LIN {X 0,Y 395.262,Z 435.098,A -85,B 0,C 180,E1 17057.331,E2 17057.331} C_VEL
LIN {X 0,Y 390.739,Z 495.427,A -85,B 0,C 180,E1 17055.904,E2 17055.904} C_VEL
LIN {X 0,Y 384.657,Z 560.923,A -85,B 0,C 180,E1 17054.093,E2 17054.093} C_VEL
LIN {X 0,Y 381.336,Z 596.706,A -85,B 0,C 180,E1 17052.908,E2 17052.908} C_VEL
LIN {X 0,Y 379.095,Z 616.56,A -85,B 0,C 180,E1 17051.979,E2 17051.979} C_VEL
LIN {X 0,Y 376.209,Z 636.469,A -85,B 0,C 180,E1 17050.759,E2 17050.759} C_VEL
LIN {X 0,Y 372.83,Z 655.705,A -85,B 0,C 180,E1 17049.265,E2 17049.265} C_VEL
LIN {X 0,Y 369.199,Z 673.643,A -85,B 0,C 180,E1 17047.542,E2 17047.542} C_VEL
LIN {X 0,Y 365.244,Z 691.251,A -85,B 0,C 180,E1 17045.476,E2 17045.476} C_VEL
LIN {X 0,Y 361.397,Z 707.145,A -85,B 0,C 180,E1 17043.216,E2 17043.216} C_VEL
LIN {X 0,Y 357.759,Z 721.542,A -85,B 0,C 180,E1 17040.76,E2 17040.76} C_VEL
LIN {X 0,Y 354.442,Z 734.528,A -85,B 0,C 180,E1 17038.106,E2 17038.106} C_VEL
LIN {X 0,Y 353.671,Z 737.462,A -85,B 0,C 180,E1 17037.421,E2 17037.421} C_VEL
LIN {X 0,Y 351.666,Z 741.92,A -85,B 0,C 180,E1 17036.434,E2 17036.434} C_VEL
LIN {X 0,Y 343.491,Z 752.769,A -85,B 0,C 180,E1 17033.979,E2 17033.979} C_VEL
LIN {X 0,Y 341.66,Z 756.437,A -85,B 0,C 180,E1 17032.885,E2 17032.885} C_VEL
LIN {X 0,Y 339.571,Z 765.333,A -85,B 0,C 180,E1 17029.568,E2 17029.568} C_VEL
LIN {X 0,Y 338.136,Z 772.212,A -85,B 0,C 180,E1 17026.315,E2 17026.315} C_VEL
LIN {X 0,Y 337.239,Z 777.506,A -85,B 0,C 180,E1 17023.022,E2 17023.022} C_VEL
LIN {X 0,Y 336.721,Z 781.379,A -85,B 0,C 180,E1 17019.572,E2 17019.572} C_VEL
LIN {X 0,Y 336.488,Z 783.588,A -85,B 0,C 180,E1 17016.141,E2 17016.141} C_VEL
LIN {X 0,Y 336.423,Z 784.209,A -85,B 0,C 180,E1 17012.896,E2 17012.896} C_VEL
LIN {X 0,Y 336.482,Z 783.288,A -85,B 0,C 180,E1 17009.489,E2 17009.489} C_VEL
LIN {X 0,Y 336.698,Z 780.724,A -85,B 0,C 180,E1 17006.084,E2 17006.084} C_VEL
LIN {X 0,Y 337.201,Z 776.517,A -85,B 0,C 180,E1 17002.675,E2 17002.675} C_VEL
LIN {X 0,Y 338.065,Z 770.919,A -85,B 0,C 180,E1 16999.434,E2 16999.434} C_VEL
LIN {X 0,Y 339.443,Z 763.662,A -85,B 0,C 180,E1 16996.196,E2 16996.196} C_VEL
LIN {X 0,Y 341.411,Z 754.589,A -85,B 0,C 180,E1 16992.971,E2 16992.971} C_VEL
LIN {X 0,Y 343.953,Z 743.864,A -85,B 0,C 180,E1 16989.878,E2 16989.878} C_VEL
LIN {X 0,Y 347.043,Z 731.447,A -85,B 0,C 180,E1 16986.932,E2 16986.932} C_VEL
LIN {X 0,Y 350.403,Z 718.053,A -85,B 0,C 180,E1 16984.296,E2 16984.296} C_VEL
LIN {X 0,Y 354.037,Z 703.239,A -85,B 0,C 180,E1 16981.859,E2 16981.859} C_VEL
LIN {X 0,Y 357.872,Z 686.847,A -85,B 0,C 180,E1 16979.622,E2 16979.622} C_VEL
LIN {X 0,Y 361.536,Z 669.791,A -85,B 0,C 180,E1 16977.693,E2 16977.693} C_VEL
LIN {X 0,Y 365.122,Z 651.237,A -85,B 0,C 180,E1 16975.977,E2 16975.977} C_VEL
LIN {X 0,Y 368.27,Z 632.306,A -85,B 0,C 180,E1 16974.564,E2 16974.564} C_VEL
LIN {X 0,Y 370.972,Z 612.338,A -85,B 0,C 180,E1 16973.39,E2 16973.39} C_VEL
LIN {X 0,Y 373.069,Z 592.248,A -85,B 0,C 180,E1 16972.505,E2 16972.505} C_VEL
LIN {X 0,Y 377.322,Z 546.729,A -85,B 0,C 180,E1 16971.047,E2 16971.047} C_VEL
LIN {X 0,Y 382.861,Z 484.443,A -85,B 0,C 180,E1 16969.345,E2 16969.345} C_VEL
LIN {X 0,Y 387.038,Z 425.627,A -85,B 0,C 180,E1 16967.978,E2 16967.978} C_VEL
LIN {X 0,Y 389.904,Z 364.859,A -85,B 0,C 180,E1 16966.743,E2 16966.743} C_VEL
LIN {X 0,Y 386.088,Z 359.453,A -85,B 0,C 180,E1 16965.944,E2 16965.944} C_VEL
LIN {X 0,Y 380.964,Z 347.137,A -85,B 0,C 180,E1 16962.826,E2 16962.826} C_VEL
LIN {X 0,Y 376.081,Z 336.257,A -85,B 0,C 180,E1 16959.649,E2 16959.649} C_VEL
LIN {X 0,Y 371.792,Z 327.479,A -85,B 0,C 180,E1 16956.658,E2 16956.658} C_VEL
LIN {X 0,Y 370.912,Z 327.517,A -85,B 0,C 180,E1 16956.374,E2 16956.374} C_VEL
LIN {X 0,Y 365.817,Z 329.462,A -85,B 0,C 180,E1 16955.029,E2 16955.029} C_VEL
LIN {X 0,Y 361.614,Z 332.459,A -85,B 0,C 180,E1 16954.146,E2 16954.146} C_VEL
LIN {X 0,Y 358.196,Z 335.591,A -85,B 0,C 180,E1 16953.553,E2 16953.553} C_VEL
LIN {X 0,Y 355.928,Z 336.945,A -85,B 0,C 180,E1 16952.918,E2 16952.918} C_VEL
LIN {X 0,Y 353.668,Z 378.738,A -85,B 0,C 180,E1 16948.911,E2 16948.911} C_VEL
LIN {X 0,Y 351.265,Z 423.605,A -85,B 0,C 180,E1 16944.646,E2 16944.646} C_VEL
LIN {X 0,Y 349.262,Z 462.521,A -85,B 0,C 180,E1 16940.969,E2 16940.969} C_VEL
LIN {X 0,Y 348.83,Z 465.633,A -85,B 0,C 180,E1 16940.754,E2 16940.754} C_VEL
LIN {X 0,Y 344.684,Z 603.323,A -85,B 0,C 180,E1 16937.135,E2 16937.135} C_VEL
LIN {X 0,Y 344.407,Z 621.566,A -85,B 0,C 180,E1 16936.464,E2 16936.464} C_VEL
LIN {X 0,Y 343.813,Z 639.774,A -85,B 0,C 180,E1 16935.433,E2 16935.433} C_VEL
LIN {X 0,Y 343.002,Z 656.912,A -85,B 0,C 180,E1 16934.088,E2 16934.088} C_VEL
LIN {X 0,Y 342.154,Z 671.753,A -85,B 0,C 180,E1 16932.568,E2 16932.568} C_VEL
LIN {X 0,Y 341.302,Z 684.893,A -85,B 0,C 180,E1 16930.892,E2 16930.892} C_VEL
LIN {X 0,Y 340.457,Z 697.128,A -85,B 0,C 180,E1 16928.955,E2 16928.955} C_VEL
LIN {X 0,Y 339.765,Z 707.457,A -85,B 0,C 180,E1 16926.931,E2 16926.931} C_VEL
LIN {X 0,Y 339.191,Z 717.119,A -85,B 0,C 180,E1 16924.566,E2 16924.566} C_VEL
LIN {X 0,Y 338.818,Z 725.023,A -85,B 0,C 180,E1 16922.03,E2 16922.03} C_VEL
LIN {X 0,Y 338.66,Z 730.537,A -85,B 0,C 180,E1 16919.662,E2 16919.662} C_VEL
LIN {X 0,Y 338.71,Z 734.833,A -85,B 0,C 180,E1 16916.955,E2 16916.955} C_VEL
LIN {X 0,Y 338.938,Z 736.969,A -85,B 0,C 180,E1 16914.414,E2 16914.414} C_VEL
LIN {X 0,Y 339.382,Z 737.372,A -85,B 0,C 180,E1 16911.85,E2 16911.85} C_VEL
LIN {X 0,Y 340.004,Z 735.908,A -85,B 0,C 180,E1 16909.324,E2 16909.324} C_VEL
LIN {X 0,Y 340.843,Z 732.779,A -85,B 0,C 180,E1 16906.887,E2 16906.887} C_VEL
LIN {X 0,Y 341.921,Z 727.575,A -85,B 0,C 180,E1 16904.394,E2 16904.394} C_VEL
LIN {X 0,Y 343.104,Z 721.104,A -85,B 0,C 180,E1 16902.183,E2 16902.183} C_VEL
LIN {X 0,Y 344.485,Z 712.486,A -85,B 0,C 180,E1 16899.972,E2 16899.972} C_VEL
LIN {X 0,Y 345.876,Z 702.622,A -85,B 0,C 180,E1 16898.007,E2 16898.007} C_VEL
LIN {X 0,Y 347.304,Z 690.717,A -85,B 0,C 180,E1 16896.142,E2 16896.142} C_VEL
LIN {X 0,Y 348.601,Z 677.563,A -85,B 0,C 180,E1 16894.518,E2 16894.518} C_VEL
LIN {X 0,Y 349.742,Z 662.299,A -85,B 0,C 180,E1 16893.056,E2 16893.056} C_VEL
LIN {X 0,Y 350.573,Z 646.797,A -85,B 0,C 180,E1 16891.928,E2 16891.928} C_VEL
LIN {X 0,Y 351.092,Z 630.054,A -85,B 0,C 180,E1 16891.038,E2 16891.038} C_VEL
LIN {X 0,Y 352.008,Z 597.232,A -85,B 0,C 180,E1 16889.859,E2 16889.859} C_VEL
LIN {X 0,Y 358.318,Z 513.728,A -85,B 0,C 180,E1 16887.077,E2 16887.077} C_VEL
LIN {X 0,Y 360.474,Z 491.875,A -85,B 0,C 180,E1 16886.307,E2 16886.307} C_VEL
LIN {X 0,Y 363.78,Z 479.698,A -85,B 0,C 180,E1 16885.515,E2 16885.515} C_VEL
LIN {X 0,Y 366.437,Z 478.721,A -85,B 0,C 180,E1 16885.216,E2 16885.216} C_VEL
LIN {X 0,Y 370.915,Z 475.814,A -85,B 0,C 180,E1 16884.864,E2 16884.864} C_VEL
LIN {X 0,Y 374.886,Z 474.256,A -85,B 0,C 180,E1 16884.45,E2 16884.45} C_VEL
LIN {X 0,Y 377.753,Z 472.722,A -85,B 0,C 180,E1 16884.201,E2 16884.201} C_VEL
LIN {X 0,Y 396.698,Z 464.403,A -85,B 0,C 180,E1 16882.483,E2 16882.483} C_VEL
LIN {X 0,Y 402.924,Z 480.075,A -85,B 0,C 180,E1 16880.192,E2 16880.192} C_VEL
LIN {X 0,Y 407.395,Z 488.925,A -85,B 0,C 180,E1 16878.854,E2 16878.854} C_VEL
LIN {X 0,Y 395.273,Z 512.025,A -85,B 0,C 180,E1 16878.047,E2 16878.047} C_VEL
LIN {X 0,Y 390.931,Z 521.783,A -85,B 0,C 180,E1 16877.657,E2 16877.657} C_VEL
LIN {X 0,Y 386.492,Z 551.571,A -85,B 0,C 180,E1 16877.527,E2 16877.527} C_VEL
LIN {X 0,Y 384.035,Z 573.78,A -85,B 0,C 180,E1 16877.191,E2 16877.191} C_VEL
LIN {X 0,Y 381.047,Z 603.773,A -85,B 0,C 180,E1 16876.316,E2 16876.316} C_VEL
LIN {X 0,Y 377.367,Z 630.176,A -85,B 0,C 180,E1 16875.298,E2 16875.298} C_VEL
LIN {X 0,Y 373.423,Z 655.596,A -85,B 0,C 180,E1 16874.014,E2 16874.014} C_VEL
LIN {X 0,Y 369.301,Z 679.477,A -85,B 0,C 180,E1 16872.494,E2 16872.494} C_VEL
LIN {X 0,Y 364.889,Z 703.359,A -85,B 0,C 180,E1 16870.622,E2 16870.622} C_VEL
LIN {X 0,Y 360.964,Z 723.184,A -85,B 0,C 180,E1 16868.757,E2 16868.757} C_VEL
LIN {X 0,Y 356.93,Z 741.602,A -85,B 0,C 180,E1 16866.632,E2 16866.632} C_VEL
LIN {X 0,Y 353.156,Z 757.77,A -85,B 0,C 180,E1 16864.391,E2 16864.391} C_VEL
LIN {X 0,Y 349.271,Z 773.512,A -85,B 0,C 180,E1 16861.765,E2 16861.765} C_VEL
LIN {X 0,Y 345.911,Z 787.154,A -85,B 0,C 180,E1 16859.052,E2 16859.052} C_VEL
LIN {X 0,Y 342.775,Z 800.117,A -85,B 0,C 180,E1 16855.947,E2 16855.947} C_VEL
LIN {X 0,Y 340.23,Z 811.492,A -85,B 0,C 180,E1 16852.666,E2 16852.666} C_VEL
LIN {X 0,Y 338.223,Z 821.847,A -85,B 0,C 180,E1 16848.977,E2 16848.977} C_VEL
LIN {X 0,Y 337.03,Z 829.629,A -85,B 0,C 180,E1 16845.486,E2 16845.486} C_VEL
LIN {X 0,Y 336.389,Z 835.947,A -85,B 0,C 180,E1 16841.835,E2 16841.835} C_VEL
LIN {X 0,Y 336.186,Z 840.283,A -85,B 0,C 180,E1 16838.38,E2 16838.38} C_VEL
LIN {X 0,Y 336.2,Z 843.205,A -85,B 0,C 180,E1 16834.777,E2 16834.777} C_VEL
LIN {X 0,Y 336.246,Z 844.515,A -85,B 0,C 180,E1 16831.363,E2 16831.363} C_VEL
LIN {X 0,Y 336.242,Z 844.359,A -85,B 0,C 180,E1 16827.955,E2 16827.955} C_VEL
LIN {X 0,Y 336.186,Z 842.807,A -85,B 0,C 180,E1 16824.539,E2 16824.539} C_VEL
LIN {X 0,Y 336.185,Z 839.823,A -85,B 0,C 180,E1 16821.103,E2 16821.103} C_VEL
LIN {X 0,Y 336.464,Z 835.014,A -85,B 0,C 180,E1 16817.471,E2 16817.471} C_VEL
LIN {X 0,Y 337.218,Z 828.492,A -85,B 0,C 180,E1 16813.816,E2 16813.816} C_VEL
LIN {X 0,Y 338.62,Z 819.993,A -85,B 0,C 180,E1 16810.149,E2 16810.149} C_VEL
LIN {X 0,Y 340.712,Z 809.957,A -85,B 0,C 180,E1 16806.661,E2 16806.661} C_VEL
LIN {X 0,Y 343.628,Z 797.671,A -85,B 0,C 180,E1 16803.191,E2 16803.191} C_VEL
LIN {X 0,Y 346.935,Z 784.673,A -85,B 0,C 180,E1 16800.166,E2 16800.166} C_VEL
LIN {X 0,Y 350.9,Z 769.453,A -85,B 0,C 180,E1 16797.221,E2 16797.221} C_VEL
LIN {X 0,Y 354.87,Z 753.849,A -85,B 0,C 180,E1 16794.718,E2 16794.718} C_VEL
LIN {X 0,Y 359.213,Z 736.069,A -85,B 0,C 180,E1 16792.35,E2 16792.35} C_VEL
LIN {X 0,Y 363.159,Z 718.29,A -85,B 0,C 180,E1 16790.404,E2 16790.404} C_VEL
LIN {X 0,Y 367.813,Z 695.391,A -85,B 0,C 180,E1 16788.355,E2 16788.355} C_VEL
LIN {X 0,Y 372.217,Z 672.364,A -85,B 0,C 180,E1 16786.659,E2 16786.659} C_VEL
LIN {X 0,Y 376.337,Z 648.888,A -85,B 0,C 180,E1 16785.246,E2 16785.246} C_VEL
LIN {X 0,Y 380.576,Z 622.555,A -85,B 0,C 180,E1 16784.01,E2 16784.01} C_VEL
LIN {X 0,Y 384.213,Z 595.765,A -85,B 0,C 180,E1 16783.055,E2 16783.055} C_VEL
LIN {X 0,Y 386.796,Z 570.495,A -85,B 0,C 180,E1 16782.375,E2 16782.375} C_VEL
LIN {X 0,Y 389.554,Z 549.245,A -85,B 0,C 180,E1 16782.124,E2 16782.124} C_VEL
LIN {X 0,Y 394.307,Z 520.558,A -85,B 0,C 180,E1 16782.096,E2 16782.096} C_VEL
LIN {X 0,Y 396.977,Z 515.374,A -85,B 0,C 180,E1 16781.822,E2 16781.822} C_VEL
LIN {X 0,Y 390.107,Z 499.418,A -85,B 0,C 180,E1 16779.182,E2 16779.182} C_VEL
LIN {X 0,Y 385.796,Z 482.675,A -85,B 0,C 180,E1 16776.59,E2 16776.59} C_VEL
LIN {X 0,Y 383.759,Z 463.778,A -85,B 0,C 180,E1 16773.887,E2 16773.887} C_VEL
LIN {X 0,Y 384.131,Z 443.886,A -85,B 0,C 180,E1 16771.284,E2 16771.284} C_VEL
LIN {X 0,Y 385.183,Z 433.187,A -85,B 0,C 180,E1 16769.979,E2 16769.979} C_VEL
LIN {X 0,Y 376.808,Z 437.419,A -85,B 0,C 180,E1 16769.051,E2 16769.051} C_VEL
LIN {X 0,Y 370.245,Z 440.926,A -85,B 0,C 180,E1 16768.311,E2 16768.311} C_VEL
LIN {X 0,Y 365.407,Z 443.376,A -85,B 0,C 180,E1 16767.721,E2 16767.721} C_VEL
LIN {X 0,Y 361.686,Z 445.669,A -85,B 0,C 180,E1 16767.315,E2 16767.315} C_VEL
LIN {X 0,Y 359.691,Z 446.286,A -85,B 0,C 180,E1 16766.965,E2 16766.965} C_VEL
LIN {X 0,Y 356.329,Z 497.328,A -85,B 0,C 180,E1 16762.52,E2 16762.52} C_VEL
LIN {X 0,Y 354.938,Z 517.232,A -85,B 0,C 180,E1 16760.789,E2 16760.789} C_VEL
LIN {X 0,Y 351.805,Z 533.167,A -85,B 0,C 180,E1 16759.724,E2 16759.724} C_VEL
LIN {X 0,Y 347.579,Z 622.76,A -85,B 0,C 180,E1 16757.057,E2 16757.057} C_VEL
LIN {X 0,Y 347.403,Z 647.348,A -85,B 0,C 180,E1 16756.21,E2 16756.21} C_VEL
LIN {X 0,Y 347.128,Z 661.31,A -85,B 0,C 180,E1 16755.452,E2 16755.452} C_VEL
LIN {X 0,Y 346.495,Z 675.527,A -85,B 0,C 180,E1 16754.368,E2 16754.368} C_VEL
LIN {X 0,Y 345.645,Z 688.486,A -85,B 0,C 180,E1 16753.04,E2 16753.04} C_VEL
LIN {X 0,Y 344.612,Z 700.346,A -85,B 0,C 180,E1 16751.463,E2 16751.463} C_VEL
LIN {X 0,Y 343.514,Z 710.48,A -85,B 0,C 180,E1 16749.719,E2 16749.719} C_VEL
LIN {X 0,Y 342.363,Z 719.365,A -85,B 0,C 180,E1 16747.72,E2 16747.72} C_VEL
LIN {X 0,Y 341.359,Z 726.103,A -85,B 0,C 180,E1 16745.715,E2 16745.715} C_VEL
LIN {X 0,Y 340.463,Z 731.409,A -85,B 0,C 180,E1 16743.535,E2 16743.535} C_VEL
LIN {X 0,Y 339.707,Z 735.075,A -85,B 0,C 180,E1 16741.18,E2 16741.18} C_VEL
LIN {X 0,Y 339.156,Z 736.807,A -85,B 0,C 180,E1 16738.817,E2 16738.817} C_VEL
LIN {X 0,Y 338.824,Z 736.811,A -85,B 0,C 180,E1 16736.616,E2 16736.616} C_VEL
LIN {X 0,Y 338.63,Z 735.051,A -85,B 0,C 180,E1 16734.238,E2 16734.238} C_VEL
LIN {X 0,Y 338.623,Z 731.425,A -85,B 0,C 180,E1 16731.851,E2 16731.851} C_VEL
LIN {X 0,Y 338.78,Z 726.28,A -85,B 0,C 180,E1 16729.628,E2 16729.628} C_VEL
LIN {X 0,Y 339.137,Z 719.167,A -85,B 0,C 180,E1 16727.39,E2 16727.39} C_VEL
LIN {X 0,Y 339.638,Z 710.594,A -85,B 0,C 180,E1 16725.334,E2 16725.334} C_VEL
LIN {X 0,Y 340.295,Z 699.689,A -85,B 0,C 180,E1 16723.309,E2 16723.309} C_VEL
LIN {X 0,Y 340.999,Z 687.441,A -85,B 0,C 180,E1 16721.538,E2 16721.538} C_VEL
LIN {X 0,Y 341.693,Z 673.472,A -85,B 0,C 180,E1 16719.978,E2 16719.978} C_VEL
LIN {X 0,Y 342.278,Z 658.595,A -85,B 0,C 180,E1 16718.728,E2 16718.728} C_VEL
LIN {X 0,Y 342.672,Z 642.965,A -85,B 0,C 180,E1 16717.787,E2 16717.787} C_VEL
LIN {X 0,Y 342.816,Z 626.752,A -85,B 0,C 180,E1 16717.158,E2 16717.158} C_VEL
LIN {X 0,Y 344.277,Z 553.681,A -85,B 0,C 180,E1 16715.281,E2 16715.281} C_VEL
LIN {X 0,Y 345.459,Z 515.015,A -85,B 0,C 180,E1 16714.268,E2 16714.268} C_VEL
LIN {X 0,Y 346.748,Z 505.237,A -85,B 0,C 180,E1 16713.451,E2 16713.451} C_VEL
LIN {X 0,Y 349.159,Z 454.821,A -85,B 0,C 180,E1 16708.972,E2 16708.972} C_VEL
LIN {X 0,Y 350.456,Z 430.233,A -85,B 0,C 180,E1 16706.76,E2 16706.76} C_VEL
LIN {X 0,Y 351.4,Z 430.726,A -85,B 0,C 180,E1 16706.495,E2 16706.495} C_VEL
LIN {X 0,Y 353.428,Z 429.366,A -85,B 0,C 180,E1 16706.031,E2 16706.031} C_VEL
LIN {X 0,Y 356.886,Z 424.461,A -85,B 0,C 180,E1 16705.362,E2 16705.362} C_VEL
LIN {X 0,Y 360.47,Z 417.488,A -85,B 0,C 180,E1 16704.763,E2 16704.763} C_VEL
LIN {X 0,Y 363.667,Z 415.265,A -85,B 0,C 180,E1 16704.104,E2 16704.104} C_VEL
LIN {X 0,Y 367.638,Z 410.202,A -85,B 0,C 180,E1 16703.395,E2 16703.395} C_VEL
LIN {X 0,Y 371.342,Z 403.874,A -85,B 0,C 180,E1 16702.808,E2 16702.808} C_VEL
LIN {X 0,Y 375.559,Z 400.244,A -85,B 0,C 180,E1 16702.047,E2 16702.047} C_VEL
LIN {X 0,Y 380.245,Z 393.951,A -85,B 0,C 180,E1 16701.305,E2 16701.305} C_VEL
LIN {X 0,Y 382.215,Z 390.931,A -85,B 0,C 180,E1 16701.013,E2 16701.013} C_VEL
LIN {X 0,Y 385.86,Z 388.381,A -85,B 0,C 180,E1 16700.397,E2 16700.397} C_VEL
LIN {X 0,Y 392.847,Z 384.511,A -85,B 0,C 180,E1 16699.244,E2 16699.244} C_VEL
LIN {X 0,Y 389.535,Z 442.145,A -85,B 0,C 180,E1 16698.061,E2 16698.061} C_VEL
LIN {X 0,Y 384.71,Z 502.485,A -85,B 0,C 180,E1 16696.594,E2 16696.594} C_VEL
LIN {X 0,Y 378.36,Z 566.803,A -85,B 0,C 180,E1 16694.764,E2 16694.764} C_VEL
LIN {X 0,Y 375.104,Z 600.539,A -85,B 0,C 180,E1 16693.588,E2 16693.588} C_VEL
LIN {X 0,Y 372.552,Z 621.211,A -85,B 0,C 180,E1 16692.557,E2 16692.557} C_VEL
LIN {X 0,Y 369.526,Z 640.385,A -85,B 0,C 180,E1 16691.317,E2 16691.317} C_VEL
LIN {X 0,Y 366.104,Z 658.655,A -85,B 0,C 180,E1 16689.835,E2 16689.835} C_VEL
LIN {X 0,Y 362.324,Z 676.277,A -85,B 0,C 180,E1 16688.081,E2 16688.081} C_VEL
LIN {X 0,Y 358.368,Z 692.96,A -85,B 0,C 180,E1 16686.065,E2 16686.065} C_VEL
LIN {X 0,Y 354.353,Z 708.694,A -85,B 0,C 180,E1 16683.771,E2 16683.771} C_VEL
LIN {X 0,Y 350.548,Z 722.959,A -85,B 0,C 180,E1 16681.273,E2 16681.273} C_VEL
LIN {X 0,Y 346.964,Z 736.185,A -85,B 0,C 180,E1 16678.485,E2 16678.485} C_VEL
LIN {X 0,Y 343.834,Z 747.923,A -85,B 0,C 180,E1 16675.492,E2 16675.492} C_VEL
LIN {X 0,Y 341.66,Z 756.437,A -85,B 0,C 180,E1 16672.885,E2 16672.885} C_VEL
LIN {X 0,Y 339.898,Z 760.008,A -85,B 0,C 180,E1 16671.763,E2 16671.763} C_VEL
LIN {X 0,Y 332.317,Z 768.392,A -85,B 0,C 180,E1 16668.918,E2 16668.918} C_VEL
LIN {X 0,Y 330.749,Z 771.047,A -85,B 0,C 180,E1 16667.684,E2 16667.684} C_VEL
LIN {X 0,Y 329.577,Z 776.981,A -85,B 0,C 180,E1 16664.225,E2 16664.225} C_VEL
LIN {X 0,Y 328.901,Z 781.297,A -85,B 0,C 180,E1 16660.687,E2 16660.687} C_VEL
LIN {X 0,Y 328.58,Z 783.91,A -85,B 0,C 180,E1 16657.167,E2 16657.167} C_VEL
LIN {X 0,Y 328.463,Z 784.88,A -85,B 0,C 180,E1 16653.84,E2 16653.84} C_VEL
LIN {X 0,Y 328.479,Z 784.354,A -85,B 0,C 180,E1 16650.349,E2 16650.349} C_VEL
LIN {X 0,Y 328.661,Z 782.234,A -85,B 0,C 180,E1 16646.861,E2 16646.861} C_VEL
LIN {X 0,Y 329.116,Z 778.49,A -85,B 0,C 180,E1 16643.371,E2 16643.371} C_VEL
LIN {X 0,Y 329.981,Z 773.047,A -85,B 0,C 180,E1 16639.878,E2 16639.878} C_VEL
LIN {X 0,Y 331.331,Z 766.206,A -85,B 0,C 180,E1 16636.564,E2 16636.564} C_VEL
LIN {X 0,Y 333.286,Z 757.573,A -85,B 0,C 180,E1 16633.262,E2 16633.262} C_VEL
LIN {X 0,Y 335.928,Z 746.919,A -85,B 0,C 180,E1 16629.984,E2 16629.984} C_VEL
LIN {X 0,Y 338.931,Z 735.458,A -85,B 0,C 180,E1 16627.082,E2 16627.082} C_VEL
LIN {X 0,Y 342.546,Z 721.776,A -85,B 0,C 180,E1 16624.22,E2 16624.22} C_VEL
LIN {X 0,Y 346.374,Z 707.02,A -85,B 0,C 180,E1 16621.659,E2 16621.659} C_VEL
LIN {X 0,Y 350.316,Z 691.142,A -85,B 0,C 180,E1 16619.371,E2 16619.371} C_VEL
LIN {X 0,Y 354.156,Z 674.387,A -85,B 0,C 180,E1 16617.368,E2 16617.368} C_VEL
LIN {X 0,Y 357.81,Z 656.787,A -85,B 0,C 180,E1 16615.635,E2 16615.635} C_VEL
LIN {X 0,Y 361.148,Z 638.361,A -85,B 0,C 180,E1 16614.158,E2 16614.158} C_VEL
LIN {X 0,Y 364.05,Z 619.039,A -85,B 0,C 180,E1 16612.925,E2 16612.925} C_VEL
LIN {X 0,Y 366.409,Z 598.92,A -85,B 0,C 180,E1 16611.942,E2 16611.942} C_VEL
LIN {X 0,Y 369.972,Z 561.878,A -85,B 0,C 180,E1 16610.66,E2 16610.66} C_VEL
LIN {X 0,Y 375.976,Z 499.713,A -85,B 0,C 180,E1 16608.875,E2 16608.875} C_VEL
LIN {X 0,Y 380.563,Z 441.4,A -85,B 0,C 180,E1 16607.445,E2 16607.445} C_VEL
LIN {X 0,Y 383.894,Z 381.895,A -85,B 0,C 180,E1 16606.212,E2 16606.212} C_VEL
LIN {X 0,Y 384.416,Z 368.795,A -85,B 0,C 180,E1 16605.942,E2 16605.942} C_VEL
LIN {X 0,Y 379.666,Z 362.118,A -85,B 0,C 180,E1 16604.893,E2 16604.893} C_VEL
LIN {X 0,Y 374.58,Z 349.858,A -85,B 0,C 180,E1 16601.634,E2 16601.634} C_VEL
LIN {X 0,Y 369.47,Z 338.503,A -85,B 0,C 180,E1 16598.099,E2 16598.099} C_VEL
LIN {X 0,Y 367.45,Z 334.602,A -85,B 0,C 180,E1 16596.676,E2 16596.676} C_VEL
LIN {X 0,Y 363.556,Z 336.124,A -85,B 0,C 180,E1 16595.666,E2 16595.666} C_VEL
LIN {X 0,Y 360.532,Z 338.198,A -85,B 0,C 180,E1 16595.035,E2 16595.035} C_VEL
LIN {X 0,Y 356.464,Z 341.766,A -85,B 0,C 180,E1 16594.319,E2 16594.319} C_VEL
LIN {X 0,Y 354.212,Z 343.231,A -85,B 0,C 180,E1 16593.786,E2 16593.786} C_VEL
LIN {X 0,Y 350.718,Z 346.596,A -85,B 0,C 180,E1 16593.188,E2 16593.188} C_VEL
LIN {X 0,Y 348.362,Z 348.033,A -85,B 0,C 180,E1 16592.559,E2 16592.559} C_VEL
LIN {X 0,Y 348.166,Z 348.119,A -85,B 0,C 180,E1 16592.482,E2 16592.482} C_VEL
LIN {X 0,Y 345.741,Z 391.338,A -85,B 0,C 180,E1 16588.313,E2 16588.313} C_VEL
LIN {X 0,Y 343.217,Z 436.478,A -85,B 0,C 180,E1 16583.981,E2 16583.981} C_VEL
LIN {X 0,Y 341.643,Z 463.906,A -85,B 0,C 180,E1 16581.369,E2 16581.369} C_VEL
LIN {X 0,Y 341.271,Z 466.787,A -85,B 0,C 180,E1 16581.18,E2 16581.18} C_VEL
LIN {X 0,Y 336.938,Z 603.557,A -85,B 0,C 180,E1 16577.469,E2 16577.469} C_VEL
LIN {X 0,Y 336.642,Z 622.447,A -85,B 0,C 180,E1 16576.766,E2 16576.766} C_VEL
LIN {X 0,Y 336.026,Z 640.753,A -85,B 0,C 180,E1 16575.711,E2 16575.711} C_VEL
LIN {X 0,Y 335.235,Z 657.013,A -85,B 0,C 180,E1 16574.422,E2 16574.422} C_VEL
LIN {X 0,Y 334.408,Z 671.374,A -85,B 0,C 180,E1 16572.959,E2 16572.959} C_VEL
LIN {X 0,Y 333.473,Z 685.515,A -85,B 0,C 180,E1 16571.151,E2 16571.151} C_VEL
LIN {X 0,Y 332.528,Z 698.866,A -85,B 0,C 180,E1 16568.996,E2 16568.996} C_VEL
LIN {X 0,Y 331.775,Z 709.893,A -85,B 0,C 180,E1 16566.75,E2 16566.75} C_VEL
LIN {X 0,Y 331.246,Z 718.754,A -85,B 0,C 180,E1 16564.502,E2 16564.502} C_VEL
LIN {X 0,Y 330.887,Z 726.674,A -85,B 0,C 180,E1 16561.905,E2 16561.905} C_VEL
LIN {X 0,Y 330.741,Z 732.474,A -85,B 0,C 180,E1 16559.308,E2 16559.308} C_VEL
LIN {X 0,Y 330.83,Z 736.423,A -85,B 0,C 180,E1 16556.709,E2 16556.709} C_VEL
LIN {X 0,Y 331.137,Z 738.618,A -85,B 0,C 180,E1 16553.934,E2 16553.934} C_VEL
LIN {X 0,Y 331.612,Z 738.872,A -85,B 0,C 180,E1 16551.484,E2 16551.484} C_VEL
LIN {X 0,Y 332.386,Z 737.199,A -85,B 0,C 180,E1 16548.712,E2 16548.712} C_VEL
LIN {X 0,Y 333.309,Z 733.958,A -85,B 0,C 180,E1 16546.292,E2 16546.292} C_VEL
LIN {X 0,Y 334.464,Z 728.876,A -85,B 0,C 180,E1 16543.859,E2 16543.859} C_VEL
LIN {X 0,Y 335.772,Z 722.296,A -85,B 0,C 180,E1 16541.601,E2 16541.601} C_VEL
LIN {X 0,Y 337.3,Z 713.585,A -85,B 0,C 180,E1 16539.345,E2 16539.345} C_VEL
LIN {X 0,Y 338.955,Z 702.651,A -85,B 0,C 180,E1 16537.177,E2 16537.177} C_VEL
LIN {X 0,Y 340.38,Z 691.47,A -85,B 0,C 180,E1 16535.44,E2 16535.44} C_VEL
LIN {X 0,Y 341.803,Z 678.158,A -85,B 0,C 180,E1 16533.787,E2 16533.787} C_VEL
LIN {X 0,Y 342.978,Z 663.67,A -85,B 0,C 180,E1 16532.386,E2 16532.386} C_VEL
LIN {X 0,Y 343.981,Z 646.934,A -85,B 0,C 180,E1 16531.151,E2 16531.151} C_VEL
LIN {X 0,Y 344.576,Z 629.173,A -85,B 0,C 180,E1 16530.22,E2 16530.22} C_VEL
LIN {X 0,Y 345.974,Z 593.683,A -85,B 0,C 180,E1 16528.909,E2 16528.909} C_VEL
LIN {X 0,Y 353.466,Z 507.766,A -85,B 0,C 180,E1 16525.914,E2 16525.914} C_VEL
LIN {X 0,Y 354.982,Z 494.406,A -85,B 0,C 180,E1 16525.421,E2 16525.421} C_VEL
LIN {X 0,Y 355.621,Z 492.642,A -85,B 0,C 180,E1 16525.296,E2 16525.296} C_VEL
LIN {X 0,Y 359.098,Z 490.983,A -85,B 0,C 180,E1 16524.946,E2 16524.946} C_VEL
LIN {X 0,Y 364.058,Z 486.876,A -85,B 0,C 180,E1 16524.656,E2 16524.656} C_VEL
LIN {X 0,Y 365.603,Z 485.617,A -85,B 0,C 180,E1 16524.565,E2 16524.565} C_VEL
LIN {X 0,Y 371.843,Z 482.103,A -85,B 0,C 180,E1 16524.035,E2 16524.035} C_VEL
LIN {X 0,Y 391.921,Z 473.051,A -85,B 0,C 180,E1 16522.234,E2 16522.234} C_VEL
LIN {X 0,Y 399.121,Z 489.554,A -85,B 0,C 180,E1 16519.735,E2 16519.735} C_VEL
LIN {X 0,Y 399.835,Z 491.049,A -85,B 0,C 180,E1 16519.51,E2 16519.51} C_VEL
LIN {X 0,Y 389.288,Z 511.078,A -85,B 0,C 180,E1 16518.812,E2 16518.812} C_VEL
LIN {X 0,Y 385.531,Z 519.485,A -85,B 0,C 180,E1 16518.485,E2 16518.485} C_VEL
LIN {X 0,Y 380.833,Z 550.549,A -85,B 0,C 180,E1 16518.364,E2 16518.364} C_VEL
LIN {X 0,Y 378.197,Z 573.264,A -85,B 0,C 180,E1 16518.018,E2 16518.018} C_VEL
LIN {X 0,Y 375.147,Z 602.665,A -85,B 0,C 180,E1 16517.151,E2 16517.151} C_VEL
LIN {X 0,Y 371.105,Z 630.572,A -85,B 0,C 180,E1 16516.059,E2 16516.059} C_VEL
LIN {X 0,Y 367.037,Z 655.719,A -85,B 0,C 180,E1 16514.764,E2 16514.764} C_VEL
LIN {X 0,Y 362.566,Z 680.551,A -85,B 0,C 180,E1 16513.151,E2 16513.151} C_VEL
LIN {X 0,Y 358.194,Z 703.382,A -85,B 0,C 180,E1 16511.334,E2 16511.334} C_VEL
LIN {X 0,Y 354.106,Z 723.083,A -85,B 0,C 180,E1 16509.444,E2 16509.444} C_VEL
LIN {X 0,Y 349.905,Z 741.506,A -85,B 0,C 180,E1 16507.286,E2 16507.286} C_VEL
LIN {X 0,Y 345.822,Z 758.086,A -85,B 0,C 180,E1 16504.923,E2 16504.923} C_VEL
LIN {X 0,Y 341.693,Z 774.127,A -85,B 0,C 180,E1 16502.179,E2 16502.179} C_VEL
LIN {X 0,Y 337.983,Z 788.38,A -85,B 0,C 180,E1 16499.217,E2 16499.217} C_VEL
LIN {X 0,Y 334.785,Z 801.118,A -85,B 0,C 180,E1 16496.042,E2 16496.042} C_VEL
LIN {X 0,Y 332.065,Z 812.771,A -85,B 0,C 180,E1 16492.483,E2 16492.483} C_VEL
LIN {X 0,Y 330.248,Z 821.849,A -85,B 0,C 180,E1 16489.086,E2 16489.086} C_VEL
LIN {X 0,Y 328.985,Z 829.832,A -85,B 0,C 180,E1 16485.332,E2 16485.332} C_VEL
LIN {X 0,Y 328.39,Z 835.672,A -85,B 0,C 180,E1 16481.771,E2 16481.771} C_VEL
LIN {X 0,Y 328.203,Z 840.045,A -85,B 0,C 180,E1 16478.056,E2 16478.056} C_VEL
LIN {X 0,Y 328.229,Z 842.686,A -85,B 0,C 180,E1 16474.543,E2 16474.543} C_VEL
LIN {X 0,Y 328.286,Z 843.828,A -85,B 0,C 180,E1 16471.047,E2 16471.047} C_VEL
LIN {X 0,Y 328.265,Z 843.535,A -85,B 0,C 180,E1 16467.491,E2 16467.491} C_VEL
LIN {X 0,Y 328.198,Z 841.873,A -85,B 0,C 180,E1 16464.054,E2 16464.054} C_VEL
LIN {X 0,Y 328.227,Z 838.714,A -85,B 0,C 180,E1 16460.532,E2 16460.532} C_VEL
LIN {X 0,Y 328.56,Z 833.746,A -85,B 0,C 180,E1 16456.807,E2 16456.807} C_VEL
LIN {X 0,Y 329.436,Z 827.022,A -85,B 0,C 180,E1 16453.06,E2 16453.06} C_VEL
LIN {X 0,Y 331.035,Z 818.331,A -85,B 0,C 180,E1 16449.305,E2 16449.305} C_VEL
LIN {X 0,Y 333.21,Z 808.615,A -85,B 0,C 180,E1 16445.915,E2 16445.915} C_VEL
LIN {X 0,Y 336.404,Z 796.053,A -85,B 0,C 180,E1 16442.339,E2 16442.339} C_VEL
LIN {X 0,Y 339.996,Z 782.702,A -85,B 0,C 180,E1 16439.223,E2 16439.223} C_VEL
LIN {X 0,Y 344.148,Z 767.599,A -85,B 0,C 180,E1 16436.295,E2 16436.295} C_VEL
LIN {X 0,Y 348.369,Z 751.748,A -85,B 0,C 180,E1 16433.754,E2 16433.754} C_VEL
LIN {X 0,Y 352.824,Z 734.287,A -85,B 0,C 180,E1 16431.431,E2 16431.431} C_VEL
LIN {X 0,Y 356.953,Z 716.342,A -85,B 0,C 180,E1 16429.469,E2 16429.469} C_VEL
LIN {X 0,Y 361.74,Z 693.664,A -85,B 0,C 180,E1 16427.448,E2 16427.448} C_VEL
LIN {X 0,Y 366.303,Z 670.542,A -85,B 0,C 180,E1 16425.747,E2 16425.747} C_VEL
LIN {X 0,Y 370.764,Z 646.001,A -85,B 0,C 180,E1 16424.286,E2 16424.286} C_VEL
LIN {X 0,Y 375.118,Z 619.724,A -85,B 0,C 180,E1 16423.071,E2 16423.071} C_VEL
LIN {X 0,Y 378.872,Z 592.395,A -85,B 0,C 180,E1 16422.109,E2 16422.109} C_VEL
LIN {X 0,Y 381.369,Z 569.17,A -85,B 0,C 180,E1 16421.495,E2 16421.495} C_VEL
LIN {X 0,Y 384.35,Z 547.133,A -85,B 0,C 180,E1 16421.248,E2 16421.248} C_VEL
LIN {X 0,Y 389.448,Z 517.699,A -85,B 0,C 180,E1 16421.214,E2 16421.214} C_VEL
LIN {X 0,Y 382.988,Z 501.509,A -85,B 0,C 180,E1 16418.509,E2 16418.509} C_VEL
LIN {X 0,Y 379.06,Z 484.428,A -85,B 0,C 180,E1 16415.843,E2 16415.843} C_VEL
LIN {X 0,Y 377.429,Z 465.235,A -85,B 0,C 180,E1 16413.073,E2 16413.073} C_VEL
LIN {X 0,Y 378.216,Z 445.06,A -85,B 0,C 180,E1 16410.414,E2 16410.414} C_VEL
LIN {X 0,Y 378.31,Z 442.423,A -85,B 0,C 180,E1 16410.055,E2 16410.055} C_VEL
LIN {X 0,Y 363.999,Z 450.075,A -85,B 0,C 180,E1 16408.477,E2 16408.477} C_VEL
LIN {X 0,Y 359.967,Z 452.2,A -85,B 0,C 180,E1 16407.996,E2 16407.996} C_VEL
LIN {X 0,Y 358.35,Z 453.126,A -85,B 0,C 180,E1 16407.811,E2 16407.811} C_VEL
LIN {X 0,Y 354.721,Z 455.225,A -85,B 0,C 180,E1 16407.389,E2 16407.389} C_VEL
LIN {X 0,Y 353.192,Z 455.674,A -85,B 0,C 180,E1 16407.114,E2 16407.114} C_VEL
LIN {X 0,Y 349.332,Z 509.007,A -85,B 0,C 180,E1 16402.375,E2 16402.375} C_VEL
LIN {X 0,Y 348.537,Z 518.647,A -85,B 0,C 180,E1 16401.542,E2 16401.542} C_VEL
LIN {X 0,Y 345.224,Z 535.166,A -85,B 0,C 180,E1 16400.442,E2 16400.442} C_VEL
LIN {X 0,Y 340.582,Z 624.082,A -85,B 0,C 180,E1 16397.677,E2 16397.677} C_VEL
LIN {X 0,Y 340.358,Z 648.757,A -85,B 0,C 180,E1 16396.803,E2 16396.803} C_VEL
LIN {X 0,Y 339.989,Z 663.637,A -85,B 0,C 180,E1 16395.96,E2 16395.96} C_VEL
LIN {X 0,Y 339.277,Z 677.694,A -85,B 0,C 180,E1 16394.842,E2 16394.842} C_VEL
LIN {X 0,Y 338.372,Z 690.441,A -85,B 0,C 180,E1 16393.499,E2 16393.499} C_VEL
LIN {X 0,Y 337.247,Z 702.168,A -85,B 0,C 180,E1 16391.89,E2 16391.89} C_VEL
LIN {X 0,Y 336.055,Z 712.211,A -85,B 0,C 180,E1 16390.11,E2 16390.11} C_VEL
LIN {X 0,Y 334.821,Z 721.076,A -85,B 0,C 180,E1 16388.068,E2 16388.068} C_VEL
LIN {X 0,Y 333.728,Z 727.742,A -85,B 0,C 180,E1 16386.019,E2 16386.019} C_VEL
LIN {X 0,Y 332.749,Z 732.973,A -85,B 0,C 180,E1 16383.79,E2 16383.79} C_VEL
LIN {X 0,Y 331.927,Z 736.601,A -85,B 0,C 180,E1 16381.38,E2 16381.38} C_VEL
LIN {X 0,Y 331.322,Z 738.274,A -85,B 0,C 180,E1 16378.962,E2 16378.962} C_VEL
LIN {X 0,Y 330.95,Z 738.199,A -85,B 0,C 180,E1 16376.709,E2 16376.709} C_VEL
LIN {X 0,Y 330.732,Z 736.369,A -85,B 0,C 180,E1 16374.274,E2 16374.274} C_VEL
LIN {X 0,Y 330.712,Z 732.65,A -85,B 0,C 180,E1 16371.83,E2 16371.83} C_VEL
LIN {X 0,Y 330.869,Z 727.405,A -85,B 0,C 180,E1 16369.553,E2 16369.553} C_VEL
LIN {X 0,Y 331.232,Z 720.188,A -85,B 0,C 180,E1 16367.269,E2 16367.269} C_VEL
LIN {X 0,Y 331.752,Z 711.442,A -85,B 0,C 180,E1 16365.156,E2 16365.156} C_VEL
LIN {X 0,Y 332.42,Z 700.645,A -85,B 0,C 180,E1 16363.126,E2 16363.126} C_VEL
LIN {X 0,Y 333.131,Z 688.633,A -85,B 0,C 180,E1 16361.358,E2 16361.358} C_VEL
LIN {X 0,Y 333.833,Z 675.068,A -85,B 0,C 180,E1 16359.804,E2 16359.804} C_VEL
LIN {X 0,Y 334.444,Z 660.214,A -85,B 0,C 180,E1 16358.516,E2 16358.516} C_VEL
LIN {X 0,Y 334.871,Z 644.337,A -85,B 0,C 180,E1 16357.53,E2 16357.53} C_VEL
LIN {X 0,Y 335.029,Z 628.044,A -85,B 0,C 180,E1 16356.88,E2 16356.88} C_VEL
LIN {X 0,Y 336.424,Z 559.308,A -85,B 0,C 180,E1 16355.057,E2 16355.057} C_VEL
LIN {X 0,Y 337.821,Z 515.978,A -85,B 0,C 180,E1 16353.879,E2 16353.879} C_VEL
LIN {X 0,Y 339.221,Z 504.906,A -85,B 0,C 180,E1 16352.942,E2 16352.942} C_VEL
LIN {X 0,Y 341.743,Z 454.552,A -85,B 0,C 180,E1 16348.418,E2 16348.418} C_VEL
LIN {X 0,Y 341.906,Z 451.464,A -85,B 0,C 180,E1 16348.139,E2 16348.139} C_VEL
LIN {X 0,Y 343.129,Z 451.811,A -85,B 0,C 180,E1 16347.774,E2 16347.774} C_VEL
LIN {X 0,Y 345.455,Z 449.729,A -85,B 0,C 180,E1 16347.231,E2 16347.231} C_VEL
LIN {X 0,Y 349.19,Z 443.834,A -85,B 0,C 180,E1 16346.501,E2 16346.501} C_VEL
LIN {X 0,Y 351.986,Z 438.277,A -85,B 0,C 180,E1 16346.02,E2 16346.02} C_VEL
LIN {X 0,Y 355.116,Z 435.901,A -85,B 0,C 180,E1 16345.336,E2 16345.336} C_VEL
LIN {X 0,Y 359.047,Z 430.663,A -85,B 0,C 180,E1 16344.603,E2 16344.603} C_VEL
LIN {X 0,Y 362.893,Z 424.045,A -85,B 0,C 180,E1 16343.967,E2 16343.967} C_VEL
LIN {X 0,Y 367.038,Z 420.236,A -85,B 0,C 180,E1 16343.179,E2 16343.179} C_VEL
LIN {X 0,Y 371.671,Z 413.766,A -85,B 0,C 180,E1 16342.41,E2 16342.41} C_VEL
LIN {X 0,Y 373.979,Z 410.126,A -85,B 0,C 180,E1 16342.053,E2 16342.053} C_VEL
LIN {X 0,Y 378.917,Z 405.363,A -85,B 0,C 180,E1 16341.216,E2 16341.216} C_VEL
LIN {X 0,Y 384.178,Z 398.027,A -85,B 0,C 180,E1 16340.432,E2 16340.432} C_VEL
LIN {X 0,Y 386.391,Z 396.092,A -85,B 0,C 180,E1 16340.077,E2 16340.077} C_VEL
LIN {X 0,Y 387.218,Z 395.818,A -85,B 0,C 180,E1 16339.933,E2 16339.933} C_VEL
LIN {X 0,Y 383.572,Z 453.001,A -85,B 0,C 180,E1 16338.723,E2 16338.723} C_VEL
LIN {X 0,Y 378.418,Z 512.66,A -85,B 0,C 180,E1 16337.218,E2 16337.218} C_VEL
LIN {X 0,Y 371.792,Z 575.966,A -85,B 0,C 180,E1 16335.343,E2 16335.343} C_VEL
LIN {X 0,Y 368.958,Z 603.82,A -85,B 0,C 180,E1 16334.305,E2 16334.305} C_VEL
LIN {X 0,Y 366.47,Z 622.812,A -85,B 0,C 180,E1 16333.329,E2 16333.329} C_VEL
LIN {X 0,Y 363.243,Z 642.235,A -85,B 0,C 180,E1 16332.043,E2 16332.043} C_VEL
LIN {X 0,Y 359.559,Z 660.881,A -85,B 0,C 180,E1 16330.491,E2 16330.491} C_VEL
LIN {X 0,Y 355.65,Z 678.178,A -85,B 0,C 180,E1 16328.721,E2 16328.721} C_VEL
LIN {X 0,Y 351.502,Z 694.782,A -85,B 0,C 180,E1 16326.662,E2 16326.662} C_VEL
LIN {X 0,Y 347.344,Z 710.247,A -85,B 0,C 180,E1 16324.347,E2 16324.347} C_VEL
LIN {X 0,Y 343.242,Z 724.8,A -85,B 0,C 180,E1 16321.723,E2 16321.723} C_VEL
LIN {X 0,Y 339.503,Z 737.842,A -85,B 0,C 180,E1 16318.881,E2 16318.881} C_VEL
LIN {X 0,Y 336.315,Z 749.124,A -85,B 0,C 180,E1 16315.915,E2 16315.915} C_VEL
LIN {X 0,Y 333.64,Z 759.029,A -85,B 0,C 180,E1 16312.743,E2 16312.743} C_VEL
LIN {X 0,Y 331.549,Z 767.496,A -85,B 0,C 180,E1 16309.374,E2 16309.374} C_VEL
LIN {X 0,Y 330.749,Z 771.047,A -85,B 0,C 180,E1 16307.684,E2 16307.684} C_VEL
LIN {X 0,Y 329.258,Z 773.568,A -85,B 0,C 180,E1 16306.43,E2 16306.43} C_VEL
LIN {X 0,Y 322.104,Z 779.549,A -85,B 0,C 180,E1 16303.067,E2 16303.067} C_VEL
LIN {X 0,Y 321.137,Z 780.943,A -85,B 0,C 180,E1 16301.918,E2 16301.918} C_VEL
LIN {X 0,Y 320.702,Z 783.968,A -85,B 0,C 180,E1 16298.426,E2 16298.426} C_VEL
LIN {X 0,Y 320.523,Z 785.472,A -85,B 0,C 180,E1 16295.011,E2 16295.011} C_VEL
LIN {X 0,Y 320.492,Z 785.472,A -85,B 0,C 180,E1 16291.609,E2 16291.609} C_VEL
LIN {X 0,Y 320.601,Z 784.024,A -85,B 0,C 180,E1 16288.213,E2 16288.213} C_VEL
LIN {X 0,Y 320.953,Z 780.951,A -85,B 0,C 180,E1 16284.637,E2 16284.637} C_VEL
LIN {X 0,Y 321.68,Z 776.221,A -85,B 0,C 180,E1 16281.059,E2 16281.059} C_VEL
LIN {X 0,Y 322.953,Z 769.727,A -85,B 0,C 180,E1 16277.484,E2 16277.484} C_VEL
LIN {X 0,Y 324.896,Z 761.324,A -85,B 0,C 180,E1 16273.92,E2 16273.92} C_VEL
LIN {X 0,Y 327.461,Z 751.375,A -85,B 0,C 180,E1 16270.56,E2 16270.56} C_VEL
LIN {X 0,Y 330.587,Z 739.926,A -85,B 0,C 180,E1 16267.411,E2 16267.411} C_VEL
LIN {X 0,Y 334.199,Z 726.989,A -85,B 0,C 180,E1 16264.48,E2 16264.48} C_VEL
LIN {X 0,Y 338.186,Z 712.524,A -85,B 0,C 180,E1 16261.768,E2 16261.768} C_VEL
LIN {X 0,Y 342.249,Z 697.159,A -85,B 0,C 180,E1 16259.376,E2 16259.376} C_VEL
LIN {X 0,Y 346.365,Z 680.502,A -85,B 0,C 180,E1 16257.23,E2 16257.23} C_VEL
LIN {X 0,Y 350.258,Z 663.125,A -85,B 0,C 180,E1 16255.384,E2 16255.384} C_VEL
LIN {X 0,Y 353.839,Z 644.887,A -85,B 0,C 180,E1 16253.802,E2 16253.802} C_VEL
LIN {X 0,Y 357.036,Z 625.766,A -85,B 0,C 180,E1 16252.475,E2 16252.475} C_VEL
LIN {X 0,Y 359.683,Z 605.865,A -85,B 0,C 180,E1 16251.403,E2 16251.403} C_VEL
LIN {X 0,Y 362.272,Z 580.217,A -85,B 0,C 180,E1 16250.397,E2 16250.397} C_VEL
LIN {X 0,Y 368.742,Z 517.885,A -85,B 0,C 180,E1 16248.486,E2 16248.486} C_VEL
LIN {X 0,Y 373.914,Z 458.645,A -85,B 0,C 180,E1 16246.944,E2 16246.944} C_VEL
LIN {X 0,Y 377.595,Z 402.092,A -85,B 0,C 180,E1 16245.707,E2 16245.707} C_VEL
LIN {X 0,Y 378.946,Z 372.77,A -85,B 0,C 180,E1 16245.109,E2 16245.109} C_VEL
LIN {X 0,Y 373.33,Z 364.9,A -85,B 0,C 180,E1 16243.815,E2 16243.815} C_VEL
LIN {X 0,Y 368.509,Z 353.24,A -85,B 0,C 180,E1 16240.561,E2 16240.561} C_VEL
LIN {X 0,Y 363.836,Z 342.863,A -85,B 0,C 180,E1 16237.16,E2 16237.16} C_VEL
LIN {X 0,Y 363.456,Z 341.956,A -85,B 0,C 180,E1 16236.85,E2 16236.85} C_VEL
LIN {X 0,Y 361.346,Z 342.791,A -85,B 0,C 180,E1 16236.31,E2 16236.31} C_VEL
LIN {X 0,Y 358.706,Z 344.694,A -85,B 0,C 180,E1 16235.792,E2 16235.792} C_VEL
LIN {X 0,Y 354.205,Z 348.374,A -85,B 0,C 180,E1 16234.963,E2 16234.963} C_VEL
LIN {X 0,Y 352.355,Z 349.763,A -85,B 0,C 180,E1 16234.579,E2 16234.579} C_VEL
LIN {X 0,Y 348.368,Z 353.247,A -85,B 0,C 180,E1 16233.836,E2 16233.836} C_VEL
LIN {X 0,Y 346.409,Z 354.552,A -85,B 0,C 180,E1 16233.358,E2 16233.358} C_VEL
LIN {X 0,Y 343.22,Z 357.734,A -85,B 0,C 180,E1 16232.81,E2 16232.81} C_VEL
LIN {X 0,Y 340.999,Z 359.336,A -85,B 0,C 180,E1 16232.253,E2 16232.253} C_VEL
LIN {X 0,Y 340.336,Z 359.805,A -85,B 0,C 180,E1 16232.001,E2 16232.001} C_VEL
LIN {X 0,Y 337.711,Z 403.93,A -85,B 0,C 180,E1 16227.7,E2 16227.7} C_VEL
LIN {X 0,Y 335.102,Z 449.565,A -85,B 0,C 180,E1 16223.288,E2 16223.288} C_VEL
LIN {X 0,Y 334.047,Z 465.315,A -85,B 0,C 180,E1 16221.787,E2 16221.787} C_VEL
LIN {X 0,Y 333.713,Z 468.07,A -85,B 0,C 180,E1 16221.614,E2 16221.614} C_VEL
LIN {X 0,Y 329.197,Z 603.529,A -85,B 0,C 180,E1 16217.819,E2 16217.819} C_VEL
LIN {X 0,Y 328.904,Z 621.871,A -85,B 0,C 180,E1 16217.138,E2 16217.138} C_VEL
LIN {X 0,Y 328.365,Z 638.205,A -85,B 0,C 180,E1 16216.223,E2 16216.223} C_VEL
LIN {X 0,Y 327.579,Z 654.961,A -85,B 0,C 180,E1 16214.947,E2 16214.947} C_VEL
LIN {X 0,Y 326.658,Z 670.819,A -85,B 0,C 180,E1 16213.362,E2 16213.362} C_VEL
LIN {X 0,Y 325.677,Z 685.318,A -85,B 0,C 180,E1 16211.512,E2 16211.512} C_VEL
LIN {X 0,Y 324.797,Z 697.553,A -85,B 0,C 180,E1 16209.57,E2 16209.57} C_VEL
LIN {X 0,Y 324.04,Z 708.433,A -85,B 0,C 180,E1 16207.447,E2 16207.447} C_VEL
LIN {X 0,Y 323.442,Z 717.867,A -85,B 0,C 180,E1 16205.144,E2 16205.144} C_VEL
LIN {X 0,Y 323.042,Z 725.923,A -85,B 0,C 180,E1 16202.662,E2 16202.662} C_VEL
LIN {X 0,Y 322.842,Z 732.752,A -85,B 0,C 180,E1 16199.823,E2 16199.823} C_VEL
LIN {X 0,Y 322.895,Z 737.112,A -85,B 0,C 180,E1 16197.161,E2 16197.161} C_VEL
LIN {X 0,Y 323.175,Z 739.73,A -85,B 0,C 180,E1 16194.497,E2 16194.497} C_VEL
LIN {X 0,Y 323.677,Z 740.484,A -85,B 0,C 180,E1 16191.831,E2 16191.831} C_VEL
LIN {X 0,Y 324.372,Z 739.595,A -85,B 0,C 180,E1 16189.343,E2 16189.343} C_VEL
LIN {X 0,Y 325.366,Z 736.746,A -85,B 0,C 180,E1 16186.675,E2 16186.675} C_VEL
LIN {X 0,Y 326.57,Z 732.323,A -85,B 0,C 180,E1 16184.188,E2 16184.188} C_VEL
LIN {X 0,Y 328.031,Z 725.826,A -85,B 0,C 180,E1 16181.703,E2 16181.703} C_VEL
LIN {X 0,Y 329.643,Z 717.732,A -85,B 0,C 180,E1 16179.4,E2 16179.4} C_VEL
LIN {X 0,Y 331.323,Z 708.029,A -85,B 0,C 180,E1 16177.278,E2 16177.278} C_VEL
LIN {X 0,Y 333.086,Z 696.124,A -85,B 0,C 180,E1 16175.245,E2 16175.245} C_VEL
LIN {X 0,Y 334.604,Z 683.546,A -85,B 0,C 180,E1 16173.562,E2 16173.562} C_VEL
LIN {X 0,Y 335.943,Z 670.162,A -85,B 0,C 180,E1 16172.124,E2 16172.124} C_VEL
LIN {X 0,Y 337.136,Z 654.114,A -85,B 0,C 180,E1 16170.8,E2 16170.8} C_VEL
LIN {X 0,Y 337.981,Z 637.071,A -85,B 0,C 180,E1 16169.753,E2 16169.753} C_VEL
LIN {X 0,Y 338.982,Z 608.975,A -85,B 0,C 180,E1 16168.585,E2 16168.585} C_VEL
LIN {X 0,Y 343.611,Z 553.614,A -85,B 0,C 180,E1 16166.568,E2 16166.568} C_VEL
LIN {X 0,Y 347.824,Z 514.026,A -85,B 0,C 180,E1 16165.107,E2 16165.107} C_VEL
LIN {X 0,Y 350.655,Z 508.834,A -85,B 0,C 180,E1 16164.707,E2 16164.707} C_VEL
LIN {X 0,Y 352.954,Z 503.485,A -85,B 0,C 180,E1 16164.449,E2 16164.449} C_VEL
LIN {X 0,Y 357.142,Z 498.786,A -85,B 0,C 180,E1 16164.35,E2 16164.35} C_VEL
LIN {X 0,Y 363.184,Z 494.731,A -85,B 0,C 180,E1 16163.904,E2 16163.904} C_VEL
LIN {X 0,Y 367.315,Z 491.3,A -85,B 0,C 180,E1 16163.682,E2 16163.682} C_VEL
LIN {X 0,Y 371.72,Z 488.699,A -85,B 0,C 180,E1 16163.335,E2 16163.335} C_VEL
LIN {X 0,Y 387.282,Z 481.702,A -85,B 0,C 180,E1 16161.961,E2 16161.961} C_VEL
LIN {X 0,Y 392.244,Z 493.127,A -85,B 0,C 180,E1 16160.205,E2 16160.205} C_VEL
LIN {X 0,Y 381.607,Z 513.785,A -85,B 0,C 180,E1 16159.45,E2 16159.45} C_VEL
LIN {X 0,Y 380.199,Z 517.304,A -85,B 0,C 180,E1 16159.336,E2 16159.336} C_VEL
LIN {X 0,Y 375.232,Z 549.718,A -85,B 0,C 180,E1 16159.224,E2 16159.224} C_VEL
LIN {X 0,Y 372.434,Z 572.851,A -85,B 0,C 180,E1 16158.869,E2 16158.869} C_VEL
LIN {X 0,Y 369.352,Z 601.267,A -85,B 0,C 180,E1 16158.02,E2 16158.02} C_VEL
LIN {X 0,Y 365.045,Z 630.156,A -85,B 0,C 180,E1 16156.882,E2 16156.882} C_VEL
LIN {X 0,Y 360.94,Z 654.5,A -85,B 0,C 180,E1 16155.619,E2 16155.619} C_VEL
LIN {X 0,Y 356.237,Z 679.837,A -85,B 0,C 180,E1 16153.965,E2 16153.965} C_VEL
LIN {X 0,Y 351.702,Z 702.629,A -85,B 0,C 180,E1 16152.139,E2 16152.139} C_VEL
LIN {X 0,Y 347.479,Z 722.232,A -85,B 0,C 180,E1 16150.24,E2 16150.24} C_VEL
LIN {X 0,Y 343.252,Z 740.08,A -85,B 0,C 180,E1 16148.137,E2 16148.137} C_VEL
LIN {X 0,Y 338.951,Z 756.794,A -85,B 0,C 180,E1 16145.738,E2 16145.738} C_VEL
LIN {X 0,Y 334.731,Z 772.485,A -85,B 0,C 180,E1 16143.034,E2 16143.034} C_VEL
LIN {X 0,Y 330.893,Z 786.522,A -85,B 0,C 180,E1 16140.106,E2 16140.106} C_VEL
LIN {X 0,Y 327.45,Z 799.47,A -85,B 0,C 180,E1 16136.867,E2 16136.867} C_VEL
LIN {X 0,Y 324.612,Z 810.854,A -85,B 0,C 180,E1 16133.382,E2 16133.382} C_VEL
LIN {X 0,Y 322.516,Z 820.556,A -85,B 0,C 180,E1 16129.75,E2 16129.75} C_VEL
LIN {X 0,Y 321.129,Z 828.665,A -85,B 0,C 180,E1 16125.902,E2 16125.902} C_VEL
LIN {X 0,Y 320.45,Z 834.644,A -85,B 0,C 180,E1 16122.25,E2 16122.25} C_VEL
LIN {X 0,Y 320.223,Z 839.115,A -85,B 0,C 180,E1 16118.439,E2 16118.439} C_VEL
LIN {X 0,Y 320.253,Z 841.844,A -85,B 0,C 180,E1 16114.836,E2 16114.836} C_VEL
LIN {X 0,Y 320.307,Z 843.076,A -85,B 0,C 180,E1 16111.431,E2 16111.431} C_VEL
LIN {X 0,Y 320.301,Z 842.984,A -85,B 0,C 180,E1 16108.032,E2 16108.032} C_VEL
LIN {X 0,Y 320.231,Z 841.494,A -85,B 0,C 180,E1 16104.445,E2 16104.445} C_VEL
LIN {X 0,Y 320.234,Z 838.388,A -85,B 0,C 180,E1 16100.656,E2 16100.656} C_VEL
LIN {X 0,Y 320.557,Z 833.57,A -85,B 0,C 180,E1 16096.838,E2 16096.838} C_VEL
LIN {X 0,Y 321.443,Z 827.008,A -85,B 0,C 180,E1 16092.999,E2 16092.999} C_VEL
LIN {X 0,Y 322.984,Z 818.943,A -85,B 0,C 180,E1 16089.334,E2 16089.334} C_VEL
LIN {X 0,Y 325.474,Z 808.408,A -85,B 0,C 180,E1 16085.498,E2 16085.498} C_VEL
LIN {X 0,Y 328.599,Z 796.714,A -85,B 0,C 180,E1 16082.057,E2 16082.057} C_VEL
LIN {X 0,Y 332.36,Z 783.504,A -85,B 0,C 180,E1 16078.839,E2 16078.839} C_VEL
LIN {X 0,Y 336.656,Z 768.588,A -85,B 0,C 180,E1 16075.852,E2 16075.852} C_VEL
LIN {X 0,Y 341.033,Z 753.102,A -85,B 0,C 180,E1 16073.266,E2 16073.266} C_VEL
LIN {X 0,Y 345.64,Z 735.927,A -85,B 0,C 180,E1 16070.903,E2 16070.903} C_VEL
LIN {X 0,Y 349.924,Z 718.485,A -85,B 0,C 180,E1 16068.913,E2 16068.913} C_VEL
LIN {X 0,Y 354.584,Z 697.573,A -85,B 0,C 180,E1 16066.968,E2 16066.968} C_VEL
LIN {X 0,Y 359.411,Z 674.236,A -85,B 0,C 180,E1 16065.185,E2 16065.185} C_VEL
LIN {X 0,Y 364.36,Z 648.336,A -85,B 0,C 180,E1 16063.576,E2 16063.576} C_VEL
LIN {X 0,Y 368.783,Z 622.954,A -85,B 0,C 180,E1 16062.355,E2 16062.355} C_VEL
LIN {X 0,Y 373.036,Z 594.133,A -85,B 0,C 180,E1 16061.294,E2 16061.294} C_VEL
LIN {X 0,Y 375.861,Z 569.337,A -85,B 0,C 180,E1 16060.617,E2 16060.617} C_VEL
LIN {X 0,Y 378.856,Z 547.6,A -85,B 0,C 180,E1 16060.365,E2 16060.365} C_VEL
LIN {X 0,Y 383.173,Z 520.546,A -85,B 0,C 180,E1 16060.325,E2 16060.325} C_VEL
LIN {X 0,Y 379.097,Z 513.06,A -85,B 0,C 180,E1 16059.395,E2 16059.395} C_VEL
LIN {X 0,Y 374.268,Z 496.855,A -85,B 0,C 180,E1 16056.73,E2 16056.73} C_VEL
LIN {X 0,Y 371.681,Z 479.161,A -85,B 0,C 180,E1 16054.023,E2 16054.023} C_VEL
LIN {X 0,Y 371.34,Z 459.942,A -85,B 0,C 180,E1 16051.309,E2 16051.309} C_VEL
LIN {X 0,Y 371.722,Z 451.728,A -85,B 0,C 180,E1 16050.198,E2 16050.198} C_VEL
LIN {X 0,Y 362.602,Z 456.67,A -85,B 0,C 180,E1 16049.213,E2 16049.213} C_VEL
LIN {X 0,Y 357.788,Z 459.231,A -85,B 0,C 180,E1 16048.658,E2 16048.658} C_VEL
LIN {X 0,Y 353.643,Z 461.508,A -85,B 0,C 180,E1 16048.174,E2 16048.174} C_VEL
LIN {X 0,Y 351.782,Z 462.628,A -85,B 0,C 180,E1 16047.967,E2 16047.967} C_VEL
LIN {X 0,Y 348.158,Z 464.711,A -85,B 0,C 180,E1 16047.539,E2 16047.539} C_VEL
LIN {X 0,Y 346.751,Z 465.133,A -85,B 0,C 180,E1 16047.288,E2 16047.288} C_VEL
LIN {X 0,Y 342.516,Z 518.757,A -85,B 0,C 180,E1 16042.437,E2 16042.437} C_VEL
LIN {X 0,Y 338.73,Z 537.342,A -85,B 0,C 180,E1 16041.192,E2 16041.192} C_VEL
LIN {X 0,Y 333.793,Z 623.366,A -85,B 0,C 180,E1 16038.422,E2 16038.422} C_VEL
LIN {X 0,Y 333.388,Z 650.355,A -85,B 0,C 180,E1 16037.423,E2 16037.423} C_VEL
LIN {X 0,Y 332.974,Z 664.969,A -85,B 0,C 180,E1 16036.574,E2 16036.574} C_VEL
LIN {X 0,Y 332.216,Z 678.969,A -85,B 0,C 180,E1 16035.447,E2 16035.447} C_VEL
LIN {X 0,Y 331.21,Z 691.814,A -85,B 0,C 180,E1 16034.064,E2 16034.064} C_VEL
LIN {X 0,Y 329.92,Z 704.073,A -85,B 0,C 180,E1 16032.336,E2 16032.336} C_VEL
LIN {X 0,Y 328.644,Z 714.073,A -85,B 0,C 180,E1 16030.517,E2 16030.517} C_VEL
LIN {X 0,Y 327.3,Z 722.822,A -85,B 0,C 180,E1 16028.431,E2 16028.431} C_VEL
LIN {X 0,Y 326.029,Z 729.893,A -85,B 0,C 180,E1 16026.161,E2 16026.161} C_VEL
LIN {X 0,Y 324.98,Z 734.909,A -85,B 0,C 180,E1 16023.881,E2 16023.881} C_VEL
LIN {X 0,Y 324.154,Z 738.141,A -85,B 0,C 180,E1 16021.59,E2 16021.59} C_VEL
LIN {X 0,Y 323.454,Z 739.799,A -85,B 0,C 180,E1 16018.937,E2 16018.937} C_VEL
LIN {X 0,Y 323.029,Z 739.425,A -85,B 0,C 180,E1 16016.45,E2 16016.45} C_VEL
LIN {X 0,Y 322.813,Z 737.227,A -85,B 0,C 180,E1 16013.954,E2 16013.954} C_VEL
LIN {X 0,Y 322.809,Z 733.15,A -85,B 0,C 180,E1 16011.449,E2 16011.449} C_VEL
LIN {X 0,Y 323.004,Z 727.541,A -85,B 0,C 180,E1 16009.115,E2 16009.115} C_VEL
LIN {X 0,Y 323.407,Z 719.854,A -85,B 0,C 180,E1 16006.774,E2 16006.774} C_VEL
LIN {X 0,Y 323.977,Z 710.55,A -85,B 0,C 180,E1 16004.608,E2 16004.608} C_VEL
LIN {X 0,Y 324.664,Z 699.62,A -85,B 0,C 180,E1 16002.618,E2 16002.618} C_VEL
LIN {X 0,Y 325.377,Z 687.607,A -85,B 0,C 180,E1 16000.896,E2 16000.896} C_VEL
LIN {X 0,Y 326.043,Z 674.784,A -85,B 0,C 180,E1 15999.451,E2 15999.451} C_VEL
LIN {X 0,Y 326.64,Z 660.423,A -85,B 0,C 180,E1 15998.21,E2 15998.21} C_VEL
LIN {X 0,Y 327.064,Z 644.923,A -85,B 0,C 180,E1 15997.243,E2 15997.243} C_VEL
LIN {X 0,Y 327.229,Z 628.883,A -85,B 0,C 180,E1 15996.592,E2 15996.592} C_VEL
LIN {X 0,Y 328.593,Z 563.944,A -85,B 0,C 180,E1 15994.803,E2 15994.803} C_VEL
LIN {X 0,Y 330.196,Z 516.835,A -85,B 0,C 180,E1 15993.471,E2 15993.471} C_VEL
LIN {X 0,Y 331.646,Z 505.8,A -85,B 0,C 180,E1 15992.53,E2 15992.53} C_VEL
LIN {X 0,Y 333.329,Z 472.956,A -85,B 0,C 180,E1 15989.539,E2 15989.539} C_VEL
LIN {X 0,Y 334.51,Z 473.18,A -85,B 0,C 180,E1 15989.161,E2 15989.161} C_VEL
LIN {X 0,Y 336.864,Z 470.899,A -85,B 0,C 180,E1 15988.581,E2 15988.581} C_VEL
LIN {X 0,Y 340.674,Z 464.687,A -85,B 0,C 180,E1 15987.812,E2 15987.812} C_VEL
LIN {X 0,Y 343.44,Z 459.329,A -85,B 0,C 180,E1 15987.312,E2 15987.312} C_VEL
LIN {X 0,Y 346.512,Z 456.795,A -85,B 0,C 180,E1 15986.604,E2 15986.604} C_VEL
LIN {X 0,Y 350.482,Z 451.276,A -85,B 0,C 180,E1 15985.83,E2 15985.83} C_VEL
LIN {X 0,Y 354.224,Z 444.751,A -85,B 0,C 180,E1 15985.187,E2 15985.187} C_VEL
LIN {X 0,Y 358.14,Z 440.998,A -85,B 0,C 180,E1 15984.401,E2 15984.401} C_VEL
LIN {X 0,Y 362.788,Z 434.367,A -85,B 0,C 180,E1 15983.594,E2 15983.594} C_VEL
LIN {X 0,Y 365.205,Z 430.359,A -85,B 0,C 180,E1 15983.208,E2 15983.208} C_VEL
LIN {X 0,Y 370.02,Z 425.574,A -85,B 0,C 180,E1 15982.349,E2 15982.349} C_VEL
LIN {X 0,Y 375.189,Z 418.263,A -85,B 0,C 180,E1 15981.542,E2 15981.542} C_VEL
LIN {X 0,Y 376.686,Z 416.207,A -85,B 0,C 180,E1 15981.31,E2 15981.31} C_VEL
LIN {X 0,Y 381.33,Z 411.664,A -85,B 0,C 180,E1 15980.551,E2 15980.551} C_VEL
LIN {X 0,Y 377.305,Z 467.539,A -85,B 0,C 180,E1 15979.31,E2 15979.31} C_VEL
LIN {X 0,Y 371.792,Z 525.884,A -85,B 0,C 180,E1 15977.769,E2 15977.769} C_VEL
LIN {X 0,Y 365.26,Z 584.937,A -85,B 0,C 180,E1 15975.935,E2 15975.935} C_VEL
LIN {X 0,Y 362.667,Z 608.676,A -85,B 0,C 180,E1 15974.97,E2 15974.97} C_VEL
LIN {X 0,Y 359.83,Z 628.235,A -85,B 0,C 180,E1 15973.891,E2 15973.891} C_VEL
LIN {X 0,Y 356.379,Z 647.308,A -85,B 0,C 180,E1 15972.544,E2 15972.544} C_VEL
LIN {X 0,Y 352.514,Z 665.521,A -85,B 0,C 180,E1 15970.935,E2 15970.935} C_VEL
LIN {X 0,Y 348.313,Z 682.863,A -85,B 0,C 180,E1 15969.057,E2 15969.057} C_VEL
LIN {X 0,Y 343.988,Z 699.061,A -85,B 0,C 180,E1 15966.932,E2 15966.932} C_VEL
LIN {X 0,Y 339.495,Z 714.78,A -85,B 0,C 180,E1 15964.435,E2 15964.435} C_VEL
LIN {X 0,Y 335.449,Z 728.319,A -85,B 0,C 180,E1 15961.842,E2 15961.842} C_VEL
LIN {X 0,Y 331.527,Z 741.262,A -85,B 0,C 180,E1 15958.852,E2 15958.852} C_VEL
LIN {X 0,Y 328.123,Z 752.67,A -85,B 0,C 180,E1 15955.64,E2 15955.64} C_VEL
LIN {X 0,Y 325.443,Z 762.118,A -85,B 0,C 180,E1 15952.365,E2 15952.365} C_VEL
LIN {X 0,Y 323.365,Z 770.154,A -85,B 0,C 180,E1 15948.883,E2 15948.883} C_VEL
LIN {X 0,Y 321.939,Z 776.517,A -85,B 0,C 180,E1 15945.307,E2 15945.307} C_VEL
LIN {X 0,Y 321.137,Z 780.943,A -85,B 0,C 180,E1 15941.918,E2 15941.918} C_VEL
LIN {X 0,Y 319.938,Z 782.432,A -85,B 0,C 180,E1 15940.571,E2 15940.571} C_VEL
LIN {X 0,Y 315.058,Z 784.82,A -85,B 0,C 180,E1 15938.022,E2 15938.022} C_VEL
LIN {X 0,Y 312.798,Z 785.77,A -85,B 0,C 180,E1 15936.343,E2 15936.343} C_VEL
LIN {X 0,Y 312.576,Z 785.994,A -85,B 0,C 180,E1 15935.732,E2 15935.732} C_VEL
LIN {X 0,Y 312.516,Z 786.26,A -85,B 0,C 180,E1 15932.2,E2 15932.2} C_VEL
LIN {X 0,Y 312.621,Z 784.982,A -85,B 0,C 180,E1 15928.534,E2 15928.534} C_VEL
LIN {X 0,Y 312.964,Z 782.107,A -85,B 0,C 180,E1 15924.868,E2 15924.868} C_VEL
LIN {X 0,Y 313.65,Z 777.861,A -85,B 0,C 180,E1 15921.383,E2 15921.383} C_VEL
LIN {X 0,Y 314.912,Z 771.676,A -85,B 0,C 180,E1 15917.718,E2 15917.718} C_VEL
LIN {X 0,Y 316.753,Z 764.073,A -85,B 0,C 180,E1 15914.248,E2 15914.248} C_VEL
LIN {X 0,Y 319.308,Z 754.585,A -85,B 0,C 180,E1 15910.805,E2 15910.805} C_VEL
LIN {X 0,Y 322.543,Z 743.285,A -85,B 0,C 180,E1 15907.487,E2 15907.487} C_VEL
LIN {X 0,Y 326.313,Z 730.452,A -85,B 0,C 180,E1 15904.403,E2 15904.403} C_VEL
LIN {X 0,Y 330.371,Z 716.488,A -85,B 0,C 180,E1 15901.63,E2 15901.63} C_VEL
LIN {X 0,Y 334.572,Z 701.555,A -85,B 0,C 180,E1 15899.168,E2 15899.168} C_VEL
LIN {X 0,Y 338.893,Z 685.091,A -85,B 0,C 180,E1 15896.919,E2 15896.919} C_VEL
LIN {X 0,Y 342.959,Z 668.136,A -85,B 0,C 180,E1 15895.008,E2 15895.008} C_VEL
LIN {X 0,Y 346.759,Z 650.241,A -85,B 0,C 180,E1 15893.354,E2 15893.354} C_VEL
LIN {X 0,Y 350.134,Z 631.712,A -85,B 0,C 180,E1 15891.973,E2 15891.973} C_VEL
LIN {X 0,Y 353.053,Z 611.796,A -85,B 0,C 180,E1 15890.809,E2 15890.809} C_VEL
LIN {X 0,Y 355.371,Z 591.104,A -85,B 0,C 180,E1 15889.91,E2 15889.91} C_VEL
LIN {X 0,Y 360.554,Z 543.338,A -85,B 0,C 180,E1 15888.322,E2 15888.322} C_VEL
LIN {X 0,Y 366.394,Z 484.641,A -85,B 0,C 180,E1 15886.667,E2 15886.667} C_VEL
LIN {X 0,Y 370.861,Z 427.58,A -85,B 0,C 180,E1 15885.312,E2 15885.312} C_VEL
LIN {X 0,Y 373.581,Z 376.78,A -85,B 0,C 180,E1 15884.258,E2 15884.258} C_VEL
LIN {X 0,Y 367.078,Z 367.801,A -85,B 0,C 180,E1 15882.707,E2 15882.707} C_VEL
LIN {X 0,Y 362.667,Z 357.044,A -85,B 0,C 180,E1 15879.559,E2 15879.559} C_VEL
LIN {X 0,Y 359.203,Z 349.412,A -85,B 0,C 180,E1 15876.96,E2 15876.96} C_VEL
LIN {X 0,Y 356.521,Z 351.495,A -85,B 0,C 180,E1 15876.482,E2 15876.482} C_VEL
LIN {X 0,Y 350.623,Z 356.116,A -85,B 0,C 180,E1 15875.373,E2 15875.373} C_VEL
LIN {X 0,Y 346.077,Z 359.838,A -85,B 0,C 180,E1 15874.491,E2 15874.491} C_VEL
LIN {X 0,Y 344.875,Z 360.727,A -85,B 0,C 180,E1 15874.226,E2 15874.226} C_VEL
LIN {X 0,Y 340.823,Z 364.439,A -85,B 0,C 180,E1 15873.473,E2 15873.473} C_VEL
LIN {X 0,Y 338.565,Z 366.056,A -85,B 0,C 180,E1 15872.916,E2 15872.916} C_VEL
LIN {X 0,Y 335.079,Z 369.577,A -85,B 0,C 180,E1 15872.286,E2 15872.286} C_VEL
LIN {X 0,Y 332.937,Z 371.094,A -85,B 0,C 180,E1 15871.706,E2 15871.706} C_VEL
LIN {X 0,Y 332.465,Z 371.493,A -85,B 0,C 180,E1 15871.51,E2 15871.51} C_VEL
LIN {X 0,Y 329.732,Z 415.876,A -85,B 0,C 180,E1 15867.154,E2 15867.154} C_VEL
LIN {X 0,Y 327.011,Z 461.871,A -85,B 0,C 180,E1 15862.66,E2 15862.66} C_VEL
LIN {X 0,Y 326.178,Z 468.857,A -85,B 0,C 180,E1 15862.074,E2 15862.074} C_VEL
LIN {X 0,Y 321.438,Z 603.825,A -85,B 0,C 180,E1 15858.159,E2 15858.159} C_VEL
LIN {X 0,Y 321.137,Z 622.212,A -85,B 0,C 180,E1 15857.471,E2 15857.471} C_VEL
LIN {X 0,Y 320.605,Z 638.273,A -85,B 0,C 180,E1 15856.572,E2 15856.572} C_VEL
LIN {X 0,Y 319.769,Z 655.75,A -85,B 0,C 180,E1 15855.228,E2 15855.228} C_VEL
LIN {X 0,Y 318.816,Z 671.731,A -85,B 0,C 180,E1 15853.605,E2 15853.605} C_VEL
LIN {X 0,Y 317.805,Z 686.367,A -85,B 0,C 180,E1 15851.709,E2 15851.709} C_VEL
LIN {X 0,Y 316.938,Z 698.21,A -85,B 0,C 180,E1 15849.809,E2 15849.809} C_VEL
LIN {X 0,Y 316.093,Z 710.052,A -85,B 0,C 180,E1 15847.452,E2 15847.452} C_VEL
LIN {X 0,Y 315.451,Z 720.107,A -85,B 0,C 180,E1 15844.91,E2 15844.91} C_VEL
LIN {X 0,Y 315.097,Z 727.495,A -85,B 0,C 180,E1 15842.547,E2 15842.547} C_VEL
LIN {X 0,Y 314.922,Z 733.977,A -85,B 0,C 180,E1 15839.819,E2 15839.819} C_VEL
LIN {X 0,Y 314.999,Z 738.478,A -85,B 0,C 180,E1 15837.09,E2 15837.09} C_VEL
LIN {X 0,Y 315.314,Z 741.191,A -85,B 0,C 180,E1 15834.359,E2 15834.359} C_VEL
LIN {X 0,Y 315.874,Z 742.041,A -85,B 0,C 180,E1 15831.628,E2 15831.628} C_VEL
LIN {X 0,Y 316.699,Z 741.108,A -85,B 0,C 180,E1 15828.897,E2 15828.897} C_VEL
LIN {X 0,Y 317.824,Z 738.245,A -85,B 0,C 180,E1 15826.168,E2 15826.168} C_VEL
LIN {X 0,Y 319.154,Z 733.732,A -85,B 0,C 180,E1 15823.624,E2 15823.624} C_VEL
LIN {X 0,Y 320.783,Z 727.234,A -85,B 0,C 180,E1 15821.086,E2 15821.086} C_VEL
LIN {X 0,Y 322.4,Z 719.74,A -85,B 0,C 180,E1 15818.916,E2 15818.916} C_VEL
LIN {X 0,Y 324.238,Z 710.213,A -85,B 0,C 180,E1 15816.752,E2 15816.752} C_VEL
LIN {X 0,Y 326.101,Z 698.729,A -85,B 0,C 180,E1 15814.725,E2 15814.725} C_VEL
LIN {X 0,Y 327.736,Z 686.931,A -85,B 0,C 180,E1 15813.061,E2 15813.061} C_VEL
LIN {X 0,Y 329.353,Z 672.38,A -85,B 0,C 180,E1 15811.436,E2 15811.436} C_VEL
LIN {X 0,Y 330.702,Z 656.482,A -85,B 0,C 180,E1 15810.076,E2 15810.076} C_VEL
LIN {X 0,Y 331.693,Z 639.192,A -85,B 0,C 180,E1 15808.972,E2 15808.972} C_VEL
LIN {X 0,Y 332.944,Z 611.154,A -85,B 0,C 180,E1 15807.738,E2 15807.738} C_VEL
LIN {X 0,Y 337.547,Z 561.4,A -85,B 0,C 180,E1 15805.834,E2 15805.834} C_VEL
LIN {X 0,Y 338.31,Z 554.999,A -85,B 0,C 180,E1 15805.582,E2 15805.582} C_VEL
LIN {X 0,Y 340.649,Z 551.707,A -85,B 0,C 180,E1 15805.249,E2 15805.249} C_VEL
LIN {X 0,Y 344.776,Z 542.242,A -85,B 0,C 180,E1 15804.792,E2 15804.792} C_VEL
LIN {X 0,Y 350.29,Z 524.241,A -85,B 0,C 180,E1 15804.288,E2 15804.288} C_VEL
LIN {X 0,Y 352.148,Z 517.787,A -85,B 0,C 180,E1 15804.13,E2 15804.13} C_VEL
LIN {X 0,Y 355.931,Z 509.989,A -85,B 0,C 180,E1 15803.65,E2 15803.65} C_VEL
LIN {X 0,Y 358.208,Z 505.656,A -85,B 0,C 180,E1 15803.411,E2 15803.411} C_VEL
LIN {X 0,Y 360.206,Z 503.505,A -85,B 0,C 180,E1 15803.36,E2 15803.36} C_VEL
LIN {X 0,Y 366.689,Z 498.855,A -85,B 0,C 180,E1 15802.944,E2 15802.944} C_VEL
LIN {X 0,Y 368.989,Z 496.978,A -85,B 0,C 180,E1 15802.824,E2 15802.824} C_VEL
LIN {X 0,Y 373.02,Z 494.746,A -85,B 0,C 180,E1 15802.506,E2 15802.506} C_VEL
LIN {X 0,Y 382.787,Z 490.403,A -85,B 0,C 180,E1 15801.658,E2 15801.658} C_VEL
LIN {X 0,Y 384.799,Z 495.143,A -85,B 0,C 180,E1 15800.921,E2 15800.921} C_VEL
LIN {X 0,Y 375.028,Z 514.71,A -85,B 0,C 180,E1 15800.21,E2 15800.21} C_VEL
LIN {X 0,Y 369.771,Z 548.48,A -85,B 0,C 180,E1 15800.113,E2 15800.113} C_VEL
LIN {X 0,Y 366.795,Z 572.103,A -85,B 0,C 180,E1 15799.753,E2 15799.753} C_VEL
LIN {X 0,Y 363.638,Z 599.908,A -85,B 0,C 180,E1 15798.915,E2 15798.915} C_VEL
LIN {X 0,Y 359.198,Z 628.939,A -85,B 0,C 180,E1 15797.769,E2 15797.769} C_VEL
LIN {X 0,Y 354.692,Z 654.573,A -85,B 0,C 180,E1 15796.425,E2 15796.425} C_VEL
LIN {X 0,Y 349.863,Z 679.776,A -85,B 0,C 180,E1 15794.763,E2 15794.763} C_VEL
LIN {X 0,Y 345.125,Z 702.567,A -85,B 0,C 180,E1 15792.908,E2 15792.908} C_VEL
LIN {X 0,Y 340.739,Z 722.177,A -85,B 0,C 180,E1 15790.983,E2 15790.983} C_VEL
LIN {X 0,Y 336.51,Z 739.297,A -85,B 0,C 180,E1 15788.934,E2 15788.934} C_VEL
LIN {X 0,Y 331.846,Z 756.595,A -85,B 0,C 180,E1 15786.411,E2 15786.411} C_VEL
LIN {X 0,Y 327.581,Z 771.766,A -85,B 0,C 180,E1 15783.746,E2 15783.746} C_VEL
LIN {X 0,Y 323.427,Z 786.214,A -85,B 0,C 180,E1 15780.67,E2 15780.67} C_VEL
LIN {X 0,Y 319.866,Z 798.934,A -85,B 0,C 180,E1 15777.41,E2 15777.41} C_VEL
LIN {X 0,Y 316.82,Z 810.543,A -85,B 0,C 180,E1 15773.765,E2 15773.765} C_VEL
LIN {X 0,Y 314.728,Z 819.671,A -85,B 0,C 180,E1 15770.26,E2 15770.26} C_VEL
LIN {X 0,Y 313.234,Z 827.835,A -85,B 0,C 180,E1 15766.314,E2 15766.314} C_VEL
LIN {X 0,Y 312.493,Z 833.852,A -85,B 0,C 180,E1 15762.567,E2 15762.567} C_VEL
LIN {X 0,Y 312.241,Z 838.355,A -85,B 0,C 180,E1 15758.656,E2 15758.656} C_VEL
LIN {X 0,Y 312.278,Z 841.108,A -85,B 0,C 180,E1 15754.959,E2 15754.959} C_VEL
LIN {X 0,Y 312.338,Z 842.355,A -85,B 0,C 180,E1 15751.467,E2 15751.467} C_VEL
LIN {X 0,Y 312.331,Z 842.273,A -85,B 0,C 180,E1 15747.982,E2 15747.982} C_VEL
LIN {X 0,Y 312.25,Z 840.785,A -85,B 0,C 180,E1 15744.303,E2 15744.303} C_VEL
LIN {X 0,Y 312.256,Z 837.73,A -85,B 0,C 180,E1 15740.478,E2 15740.478} C_VEL
LIN {X 0,Y 312.582,Z 833.125,A -85,B 0,C 180,E1 15736.685,E2 15736.685} C_VEL
LIN {X 0,Y 313.578,Z 826.266,A -85,B 0,C 180,E1 15732.559,E2 15732.559} C_VEL
LIN {X 0,Y 315.24,Z 818.188,A -85,B 0,C 180,E1 15728.803,E2 15728.803} C_VEL
LIN {X 0,Y 317.904,Z 807.616,A -85,B 0,C 180,E1 15724.875,E2 15724.875} C_VEL
LIN {X 0,Y 321.232,Z 795.904,A -85,B 0,C 180,E1 15721.358,E2 15721.358} C_VEL
LIN {X 0,Y 325.279,Z 782.469,A -85,B 0,C 180,E1 15718.035,E2 15718.035} C_VEL
LIN {X 0,Y 329.752,Z 767.694,A -85,B 0,C 180,E1 15715.034,E2 15715.034} C_VEL
LIN {X 0,Y 334.54,Z 751.59,A -85,B 0,C 180,E1 15712.323,E2 15712.323} C_VEL
LIN {X 0,Y 339.381,Z 734.242,A -85,B 0,C 180,E1 15709.929,E2 15709.929} C_VEL
LIN {X 0,Y 344.088,Z 715.795,A -85,B 0,C 180,E1 15707.836,E2 15707.836} C_VEL
LIN {X 0,Y 349.206,Z 693.392,A -85,B 0,C 180,E1 15705.797,E2 15705.797} C_VEL
LIN {X 0,Y 354.354,Z 669.151,A -85,B 0,C 180,E1 15703.985,E2 15703.985} C_VEL
LIN {X 0,Y 359.278,Z 644.017,A -85,B 0,C 180,E1 15702.482,E2 15702.482} C_VEL
LIN {X 0,Y 363.89,Z 617.856,A -85,B 0,C 180,E1 15701.266,E2 15701.266} C_VEL
LIN {X 0,Y 367.971,Z 590.15,A -85,B 0,C 180,E1 15700.274,E2 15700.274} C_VEL
LIN {X 0,Y 370.627,Z 568.06,A -85,B 0,C 180,E1 15699.687,E2 15699.687} C_VEL
LIN {X 0,Y 373.872,Z 545.282,A -85,B 0,C 180,E1 15699.439,E2 15699.439} C_VEL
LIN {X 0,Y 377.355,Z 523.505,A -85,B 0,C 180,E1 15699.415,E2 15699.415} C_VEL
LIN {X 0,Y 369.766,Z 508.503,A -85,B 0,C 180,E1 15697.572,E2 15697.572} C_VEL
LIN {X 0,Y 366.249,Z 491.247,A -85,B 0,C 180,E1 15694.789,E2 15694.789} C_VEL
LIN {X 0,Y 365.017,Z 471.736,A -85,B 0,C 180,E1 15691.879,E2 15691.879} C_VEL
LIN {X 0,Y 365.355,Z 460.912,A -85,B 0,C 180,E1 15690.371,E2 15690.371} C_VEL
LIN {X 0,Y 351.671,Z 468.43,A -85,B 0,C 180,E1 15688.872,E2 15688.872} C_VEL
LIN {X 0,Y 347.254,Z 470.925,A -85,B 0,C 180,E1 15688.365,E2 15688.365} C_VEL
LIN {X 0,Y 345.374,Z 472.066,A -85,B 0,C 180,E1 15688.156,E2 15688.156} C_VEL
LIN {X 0,Y 341.73,Z 474.164,A -85,B 0,C 180,E1 15687.723,E2 15687.723} C_VEL
LIN {X 0,Y 340.359,Z 474.779,A -85,B 0,C 180,E1 15687.465,E2 15687.465} C_VEL
LIN {X 0,Y 336.238,Z 521.257,A -85,B 0,C 180,E1 15683.204,E2 15683.204} C_VEL
LIN {X 0,Y 332.441,Z 539.243,A -85,B 0,C 180,E1 15682.007,E2 15682.007} C_VEL
LIN {X 0,Y 327.031,Z 625.364,A -85,B 0,C 180,E1 15679.121,E2 15679.121} C_VEL
LIN {X 0,Y 326.515,Z 652.654,A -85,B 0,C 180,E1 15678.056,E2 15678.056} C_VEL
LIN {X 0,Y 326.056,Z 666.686,A -85,B 0,C 180,E1 15677.212,E2 15677.212} C_VEL
LIN {X 0,Y 325.21,Z 680.527,A -85,B 0,C 180,E1 15676.063,E2 15676.063} C_VEL
LIN {X 0,Y 324.037,Z 694.005,A -85,B 0,C 180,E1 15674.564,E2 15674.564} C_VEL
LIN {X 0,Y 322.719,Z 705.611,A -85,B 0,C 180,E1 15672.889,E2 15672.889} C_VEL
LIN {X 0,Y 321.258,Z 715.968,A -85,B 0,C 180,E1 15670.943,E2 15670.943} C_VEL
LIN {X 0,Y 319.812,Z 724.649,A -85,B 0,C 180,E1 15668.811,E2 15668.811} C_VEL
LIN {X 0,Y 318.435,Z 731.629,A -85,B 0,C 180,E1 15666.49,E2 15666.49} C_VEL
LIN {X 0,Y 317.289,Z 736.537,A -85,B 0,C 180,E1 15664.156,E2 15664.156} C_VEL
LIN {X 0,Y 316.39,Z 739.701,A -85,B 0,C 180,E1 15661.81,E2 15661.81} C_VEL
LIN {X 0,Y 315.663,Z 741.229,A -85,B 0,C 180,E1 15659.273,E2 15659.273} C_VEL
LIN {X 0,Y 315.179,Z 740.893,A -85,B 0,C 180,E1 15656.726,E2 15656.726} C_VEL
LIN {X 0,Y 314.931,Z 738.964,A -85,B 0,C 180,E1 15654.351,E2 15654.351} C_VEL
LIN {X 0,Y 314.885,Z 735.054,A -85,B 0,C 180,E1 15651.784,E2 15651.784} C_VEL
LIN {X 0,Y 315.062,Z 729.085,A -85,B 0,C 180,E1 15649.208,E2 15649.208} C_VEL
LIN {X 0,Y 315.461,Z 721.427,A -85,B 0,C 180,E1 15646.808,E2 15646.808} C_VEL
LIN {X 0,Y 316.036,Z 712.173,A -85,B 0,C 180,E1 15644.587,E2 15644.587} C_VEL
LIN {X 0,Y 316.738,Z 701.306,A -85,B 0,C 180,E1 15642.548,E2 15642.548} C_VEL
LIN {X 0,Y 317.473,Z 689.393,A -85,B 0,C 180,E1 15640.784,E2 15640.784} C_VEL
LIN {X 0,Y 318.164,Z 676.62,A -85,B 0,C 180,E1 15639.295,E2 15639.295} C_VEL
LIN {X 0,Y 318.797,Z 661.951,A -85,B 0,C 180,E1 15637.988,E2 15637.988} C_VEL
LIN {X 0,Y 319.252,Z 646.339,A -85,B 0,C 180,E1 15636.984,E2 15636.984} C_VEL
LIN {X 0,Y 319.432,Z 630.152,A -85,B 0,C 180,E1 15636.307,E2 15636.307} C_VEL
LIN {X 0,Y 320.744,Z 568.333,A -85,B 0,C 180,E1 15634.551,E2 15634.551} C_VEL
LIN {X 0,Y 322.514,Z 518.073,A -85,B 0,C 180,E1 15633.087,E2 15633.087} C_VEL
LIN {X 0,Y 324.057,Z 507.002,A -85,B 0,C 180,E1 15632.136,E2 15632.136} C_VEL
LIN {X 0,Y 324.788,Z 494.47,A -85,B 0,C 180,E1 15630.95,E2 15630.95} C_VEL
LIN {X 0,Y 325.823,Z 494.541,A -85,B 0,C 180,E1 15630.593,E2 15630.593} C_VEL
LIN {X 0,Y 328.041,Z 492.368,A -85,B 0,C 180,E1 15630.008,E2 15630.008} C_VEL
LIN {X 0,Y 331.726,Z 486.355,A -85,B 0,C 180,E1 15629.223,E2 15629.223} C_VEL
LIN {X 0,Y 334.655,Z 480.666,A -85,B 0,C 180,E1 15628.676,E2 15628.676} C_VEL
LIN {X 0,Y 337.659,Z 478.061,A -85,B 0,C 180,E1 15627.941,E2 15627.941} C_VEL
LIN {X 0,Y 341.62,Z 472.41,A -85,B 0,C 180,E1 15627.134,E2 15627.134} C_VEL
LIN {X 0,Y 345.318,Z 465.82,A -85,B 0,C 180,E1 15626.474,E2 15626.474} C_VEL
LIN {X 0,Y 349.33,Z 461.835,A -85,B 0,C 180,E1 15625.627,E2 15625.627} C_VEL
LIN {X 0,Y 353.98,Z 455.037,A -85,B 0,C 180,E1 15624.789,E2 15624.789} C_VEL
LIN {X 0,Y 356.362,Z 451.019,A -85,B 0,C 180,E1 15624.394,E2 15624.394} C_VEL
LIN {X 0,Y 361.074,Z 446.153,A -85,B 0,C 180,E1 15623.51,E2 15623.51} C_VEL
LIN {X 0,Y 366.336,Z 438.507,A -85,B 0,C 180,E1 15622.655,E2 15622.655} C_VEL
LIN {X 0,Y 367.748,Z 436.413,A -85,B 0,C 180,E1 15622.431,E2 15622.431} C_VEL
LIN {X 0,Y 373.158,Z 430.741,A -85,B 0,C 180,E1 15621.515,E2 15621.515} C_VEL
LIN {X 0,Y 375.354,Z 428.07,A -85,B 0,C 180,E1 15621.168,E2 15621.168} C_VEL
LIN {X 0,Y 370.889,Z 483.164,A -85,B 0,C 180,E1 15619.877,E2 15619.877} C_VEL
LIN {X 0,Y 364.781,Z 541.84,A -85,B 0,C 180,E1 15618.245,E2 15618.245} C_VEL
LIN {X 0,Y 359.171,Z 590.303,A -85,B 0,C 180,E1 15616.658,E2 15616.658} C_VEL
LIN {X 0,Y 356.587,Z 612.199,A -85,B 0,C 180,E1 15615.72,E2 15615.72} C_VEL
LIN {X 0,Y 353.445,Z 632.342,A -85,B 0,C 180,E1 15614.553,E2 15614.553} C_VEL
LIN {X 0,Y 349.681,Z 651.751,A -85,B 0,C 180,E1 15613.109,E2 15613.109} C_VEL
LIN {X 0,Y 345.491,Z 670.113,A -85,B 0,C 180,E1 15611.398,E2 15611.398} C_VEL
LIN {X 0,Y 340.988,Z 687.508,A -85,B 0,C 180,E1 15609.408,E2 15609.408} C_VEL
LIN {X 0,Y 336.322,Z 703.9,A -85,B 0,C 180,E1 15607.122,E2 15607.122} C_VEL
LIN {X 0,Y 331.638,Z 719.214,A -85,B 0,C 180,E1 15604.528,E2 15604.528} C_VEL
LIN {X 0,Y 327.276,Z 732.986,A -85,B 0,C 180,E1 15601.701,E2 15601.701} C_VEL
LIN {X 0,Y 323.331,Z 745.277,A -85,B 0,C 180,E1 15598.641,E2 15598.641} C_VEL
LIN {X 0,Y 319.927,Z 756.104,A -85,B 0,C 180,E1 15595.351,E2 15595.351} C_VEL
LIN {X 0,Y 317.153,Z 765.426,A -85,B 0,C 180,E1 15591.84,E2 15591.84} C_VEL
LIN {X 0,Y 315.164,Z 772.85,A -85,B 0,C 180,E1 15588.305,E2 15588.305} C_VEL
LIN {X 0,Y 313.787,Z 778.802,A -85,B 0,C 180,E1 15584.58,E2 15584.58} C_VEL
LIN {X 0,Y 313.02,Z 782.991,A -85,B 0,C 180,E1 15580.863,E2 15580.863} C_VEL
LIN {X 0,Y 312.655,Z 785.5,A -85,B 0,C 180,E1 15577.165,E2 15577.165} C_VEL
LIN {X 0,Y 312.576,Z 785.994,A -85,B 0,C 180,E1 15575.732,E2 15575.732} C_VEL
LIN {X 0,Y 311.555,Z 786.415,A -85,B 0,C 180,E1 15574.323,E2 15574.323} C_VEL
LIN {X 0,Y 307.283,Z 786.716,A -85,B 0,C 180,E1 15571.852,E2 15571.852} C_VEL
LIN {X 0,Y 304.806,Z 786.395,A -85,B 0,C 180,E1 15569.91,E2 15569.91} C_VEL
LIN {X 0,Y 304.624,Z 786.167,A -85,B 0,C 180,E1 15569.281,E2 15569.281} C_VEL
LIN {X 0,Y 304.928,Z 783.612,A -85,B 0,C 180,E1 15565.486,E2 15565.486} C_VEL
LIN {X 0,Y 305.618,Z 779.428,A -85,B 0,C 180,E1 15561.724,E2 15561.724} C_VEL
LIN {X 0,Y 306.857,Z 773.529,A -85,B 0,C 180,E1 15557.963,E2 15557.963} C_VEL
LIN {X 0,Y 308.822,Z 765.79,A -85,B 0,C 180,E1 15554.219,E2 15554.219} C_VEL
LIN {X 0,Y 311.443,Z 756.545,A -85,B 0,C 180,E1 15550.69,E2 15550.69} C_VEL
LIN {X 0,Y 314.667,Z 745.862,A -85,B 0,C 180,E1 15547.388,E2 15547.388} C_VEL
LIN {X 0,Y 318.407,Z 733.784,A -85,B 0,C 180,E1 15544.32,E2 15544.32} C_VEL
LIN {X 0,Y 322.549,Z 720.306,A -85,B 0,C 180,E1 15541.485,E2 15541.485} C_VEL
LIN {X 0,Y 326.991,Z 705.389,A -85,B 0,C 180,E1 15538.885,E2 15538.885} C_VEL
LIN {X 0,Y 331.421,Z 689.508,A -85,B 0,C 180,E1 15536.593,E2 15536.593} C_VEL
LIN {X 0,Y 335.882,Z 672.049,A -85,B 0,C 180,E1 15534.516,E2 15534.516} C_VEL
LIN {X 0,Y 340.082,Z 653.533,A -85,B 0,C 180,E1 15532.724,E2 15532.724} C_VEL
LIN {X 0,Y 343.8,Z 634.25,A -85,B 0,C 180,E1 15531.233,E2 15531.233} C_VEL
LIN {X 0,Y 346.929,Z 614.018,A -85,B 0,C 180,E1 15530.014,E2 15530.014} C_VEL
LIN {X 0,Y 349.361,Z 593.472,A -85,B 0,C 180,E1 15529.091,E2 15529.091} C_VEL
LIN {X 0,Y 354.613,Z 547.257,A -85,B 0,C 180,E1 15527.509,E2 15527.509} C_VEL
LIN {X 0,Y 360.806,Z 487.902,A -85,B 0,C 180,E1 15525.803,E2 15525.803} C_VEL
LIN {X 0,Y 365.366,Z 432.323,A -85,B 0,C 180,E1 15524.462,E2 15524.462} C_VEL
LIN {X 0,Y 368.297,Z 380.82,A -85,B 0,C 180,E1 15523.382,E2 15523.382} C_VEL
LIN {X 0,Y 361.013,Z 370.861,A -85,B 0,C 180,E1 15521.6,E2 15521.6} C_VEL
LIN {X 0,Y 356.573,Z 360.127,A -85,B 0,C 180,E1 15518.266,E2 15518.266} C_VEL
LIN {X 0,Y 355.365,Z 357.434,A -85,B 0,C 180,E1 15517.326,E2 15517.326} C_VEL
LIN {X 0,Y 349.001,Z 362.429,A -85,B 0,C 180,E1 15516.17,E2 15516.17} C_VEL
LIN {X 0,Y 343.113,Z 367.151,A -85,B 0,C 180,E1 15515.036,E2 15515.036} C_VEL
LIN {X 0,Y 338.507,Z 371.074,A -85,B 0,C 180,E1 15514.14,E2 15514.14} C_VEL
LIN {X 0,Y 336.775,Z 372.466,A -85,B 0,C 180,E1 15513.767,E2 15513.767} C_VEL
LIN {X 0,Y 332.654,Z 376.263,A -85,B 0,C 180,E1 15512.959,E2 15512.959} C_VEL
LIN {X 0,Y 330.498,Z 377.917,A -85,B 0,C 180,E1 15512.428,E2 15512.428} C_VEL
LIN {X 0,Y 326.755,Z 381.716,A -85,B 0,C 180,E1 15511.715,E2 15511.715} C_VEL
LIN {X 0,Y 324.517,Z 383.172,A -85,B 0,C 180,E1 15511.019,E2 15511.019} C_VEL
LIN {X 0,Y 321.671,Z 427.877,A -85,B 0,C 180,E1 15506.591,E2 15506.591} C_VEL
LIN {X 0,Y 319.253,Z 465.878,A -85,B 0,C 180,E1 15502.853,E2 15502.853} C_VEL
LIN {X 0,Y 318.628,Z 470.087,A -85,B 0,C 180,E1 15502.535,E2 15502.535} C_VEL
LIN {X 0,Y 313.697,Z 603.742,A -85,B 0,C 180,E1 15498.527,E2 15498.527} C_VEL
LIN {X 0,Y 313.385,Z 622.46,A -85,B 0,C 180,E1 15497.824,E2 15497.824} C_VEL
LIN {X 0,Y 312.806,Z 639.349,A -85,B 0,C 180,E1 15496.863,E2 15496.863} C_VEL
LIN {X 0,Y 311.96,Z 656.415,A -85,B 0,C 180,E1 15495.524,E2 15495.524} C_VEL
LIN {X 0,Y 310.941,Z 672.99,A -85,B 0,C 180,E1 15493.805,E2 15493.805} C_VEL
LIN {X 0,Y 309.924,Z 687.253,A -85,B 0,C 180,E1 15491.916,E2 15491.916} C_VEL
LIN {X 0,Y 308.99,Z 699.715,A -85,B 0,C 180,E1 15489.876,E2 15489.876} C_VEL
LIN {X 0,Y 308.138,Z 711.593,A -85,B 0,C 180,E1 15487.458,E2 15487.458} C_VEL
LIN {X 0,Y 307.498,Z 721.688,A -85,B 0,C 180,E1 15484.85,E2 15484.85} C_VEL
LIN {X 0,Y 307.134,Z 729.566,A -85,B 0,C 180,E1 15482.24,E2 15482.24} C_VEL
LIN {X 0,Y 306.998,Z 735.923,A -85,B 0,C 180,E1 15479.441,E2 15479.441} C_VEL
LIN {X 0,Y 307.15,Z 740.537,A -85,B 0,C 180,E1 15476.455,E2 15476.455} C_VEL
LIN {X 0,Y 307.556,Z 742.96,A -85,B 0,C 180,E1 15473.655,E2 15473.655} C_VEL
LIN {X 0,Y 308.233,Z 743.619,A -85,B 0,C 180,E1 15470.855,E2 15470.855} C_VEL
LIN {X 0,Y 309.204,Z 742.367,A -85,B 0,C 180,E1 15468.057,E2 15468.057} C_VEL
LIN {X 0,Y 310.418,Z 739.527,A -85,B 0,C 180,E1 15465.45,E2 15465.45} C_VEL
LIN {X 0,Y 311.91,Z 734.838,A -85,B 0,C 180,E1 15462.848,E2 15462.848} C_VEL
LIN {X 0,Y 313.731,Z 728.144,A -85,B 0,C 180,E1 15460.256,E2 15460.256} C_VEL
LIN {X 0,Y 315.698,Z 719.763,A -85,B 0,C 180,E1 15457.86,E2 15457.86} C_VEL
LIN {X 0,Y 317.736,Z 709.761,A -85,B 0,C 180,E1 15455.655,E2 15455.655} C_VEL
LIN {X 0,Y 319.667,Z 698.682,A -85,B 0,C 180,E1 15453.732,E2 15453.732} C_VEL
LIN {X 0,Y 321.623,Z 685.447,A -85,B 0,C 180,E1 15451.903,E2 15451.903} C_VEL
LIN {X 0,Y 323.405,Z 670.055,A -85,B 0,C 180,E1 15450.251,E2 15450.251} C_VEL
LIN {X 0,Y 324.893,Z 653.075,A -85,B 0,C 180,E1 15448.868,E2 15448.868} C_VEL
LIN {X 0,Y 325.939,Z 635.232,A -85,B 0,C 180,E1 15447.806,E2 15447.806} C_VEL
LIN {X 0,Y 328.143,Z 601.654,A -85,B 0,C 180,E1 15446.34,E2 15446.34} C_VEL
LIN {X 0,Y 330.015,Z 585.065,A -85,B 0,C 180,E1 15445.648,E2 15445.648} C_VEL
LIN {X 0,Y 332.503,Z 582.215,A -85,B 0,C 180,E1 15445.314,E2 15445.314} C_VEL
LIN {X 0,Y 336.711,Z 574.361,A -85,B 0,C 180,E1 15444.929,E2 15444.929} C_VEL
LIN {X 0,Y 341.783,Z 560.755,A -85,B 0,C 180,E1 15444.611,E2 15444.611} C_VEL
LIN {X 0,Y 342.647,Z 558.844,A -85,B 0,C 180,E1 15444.53,E2 15444.53} C_VEL
LIN {X 0,Y 346.447,Z 551.944,A -85,B 0,C 180,E1 15444.085,E2 15444.085} C_VEL
LIN {X 0,Y 350.851,Z 540.533,A -85,B 0,C 180,E1 15443.66,E2 15443.66} C_VEL
LIN {X 0,Y 356.596,Z 521.276,A -85,B 0,C 180,E1 15443.178,E2 15443.178} C_VEL
LIN {X 0,Y 362.634,Z 508.821,A -85,B 0,C 180,E1 15442.459,E2 15442.459} C_VEL
LIN {X 0,Y 369.727,Z 503.417,A -85,B 0,C 180,E1 15442.032,E2 15442.032} C_VEL
LIN {X 0,Y 373.328,Z 501.206,A -85,B 0,C 180,E1 15441.781,E2 15441.781} C_VEL
LIN {X 0,Y 375.852,Z 500.206,A -85,B 0,C 180,E1 15441.552,E2 15441.552} C_VEL
LIN {X 0,Y 369.886,Z 512.474,A -85,B 0,C 180,E1 15441.108,E2 15441.108} C_VEL
LIN {X 0,Y 364.388,Z 547.348,A -85,B 0,C 180,E1 15441.027,E2 15441.027} C_VEL
LIN {X 0,Y 361.237,Z 571.469,A -85,B 0,C 180,E1 15440.662,E2 15440.662} C_VEL
LIN {X 0,Y 357.942,Z 599.092,A -85,B 0,C 180,E1 15439.82,E2 15439.82} C_VEL
LIN {X 0,Y 353.442,Z 627.737,A -85,B 0,C 180,E1 15438.683,E2 15438.683} C_VEL
LIN {X 0,Y 348.678,Z 653.837,A -85,B 0,C 180,E1 15437.311,E2 15437.311} C_VEL
LIN {X 0,Y 343.811,Z 678.519,A -85,B 0,C 180,E1 15435.677,E2 15435.677} C_VEL
LIN {X 0,Y 338.821,Z 701.624,A -85,B 0,C 180,E1 15433.79,E2 15433.79} C_VEL
LIN {X 0,Y 334.25,Z 721.356,A -85,B 0,C 180,E1 15431.842,E2 15431.842} C_VEL
LIN {X 0,Y 329.835,Z 738.482,A -85,B 0,C 180,E1 15429.764,E2 15429.764} C_VEL
LIN {X 0,Y 325.104,Z 755.293,A -85,B 0,C 180,E1 15427.292,E2 15427.292} C_VEL
LIN {X 0,Y 320.625,Z 770.569,A -85,B 0,C 180,E1 15424.581,E2 15424.581} C_VEL
LIN {X 0,Y 316.228,Z 785.121,A -85,B 0,C 180,E1 15421.447,E2 15421.447} C_VEL
LIN {X 0,Y 312.591,Z 797.445,A -85,B 0,C 180,E1 15418.255,E2 15418.255} C_VEL
LIN {X 0,Y 309.39,Z 808.879,A -85,B 0,C 180,E1 15414.639,E2 15414.639} C_VEL
LIN {X 0,Y 306.974,Z 818.76,A -85,B 0,C 180,E1 15410.805,E2 15410.805} C_VEL
LIN {X 0,Y 305.347,Z 827,A -85,B 0,C 180,E1 15406.748,E2 15406.748} C_VEL
LIN {X 0,Y 304.53,Z 833.176,A -85,B 0,C 180,E1 15402.806,E2 15402.806} C_VEL
LIN {X 0,Y 304.264,Z 837.593,A -85,B 0,C 180,E1 15398.885,E2 15398.885} C_VEL
LIN {X 0,Y 304.302,Z 840.37,A -85,B 0,C 180,E1 15395.09,E2 15395.09} C_VEL
LIN {X 0,Y 304.369,Z 841.634,A -85,B 0,C 180,E1 15391.506,E2 15391.506} C_VEL
LIN {X 0,Y 304.361,Z 841.563,A -85,B 0,C 180,E1 15387.929,E2 15387.929} C_VEL
LIN {X 0,Y 304.27,Z 840.075,A -85,B 0,C 180,E1 15384.153,E2 15384.153} C_VEL
LIN {X 0,Y 304.273,Z 837.114,A -85,B 0,C 180,E1 15380.336,E2 15380.336} C_VEL
LIN {X 0,Y 304.607,Z 832.681,A -85,B 0,C 180,E1 15376.523,E2 15376.523} C_VEL
LIN {X 0,Y 305.589,Z 826.223,A -85,B 0,C 180,E1 15372.481,E2 15372.481} C_VEL
LIN {X 0,Y 307.407,Z 817.898,A -85,B 0,C 180,E1 15368.436,E2 15368.436} C_VEL
LIN {X 0,Y 310.208,Z 807.373,A -85,B 0,C 180,E1 15364.411,E2 15364.411} C_VEL
LIN {X 0,Y 313.649,Z 795.954,A -85,B 0,C 180,E1 15360.863,E2 15360.863} C_VEL
LIN {X 0,Y 317.908,Z 782.514,A -85,B 0,C 180,E1 15357.446,E2 15357.446} C_VEL
LIN {X 0,Y 322.523,Z 768.096,A -85,B 0,C 180,E1 15354.423,E2 15354.423} C_VEL
LIN {X 0,Y 327.618,Z 751.744,A -85,B 0,C 180,E1 15351.606,E2 15351.606} C_VEL
LIN {X 0,Y 332.477,Z 735.27,A -85,B 0,C 180,E1 15349.263,E2 15349.263} C_VEL
LIN {X 0,Y 337.352,Z 717.06,A -85,B 0,C 180,E1 15347.14,E2 15347.14} C_VEL
LIN {X 0,Y 341.986,Z 697.858,A -85,B 0,C 180,E1 15345.319,E2 15345.319} C_VEL
LIN {X 0,Y 347.233,Z 674.371,A -85,B 0,C 180,E1 15343.478,E2 15343.478} C_VEL
LIN {X 0,Y 352.456,Z 649.116,A -85,B 0,C 180,E1 15341.869,E2 15341.869} C_VEL
LIN {X 0,Y 357.293,Z 623.532,A -85,B 0,C 180,E1 15340.598,E2 15340.598} C_VEL
LIN {X 0,Y 361.743,Z 595.815,A -85,B 0,C 180,E1 15339.541,E2 15339.541} C_VEL
LIN {X 0,Y 364.947,Z 570.767,A -85,B 0,C 180,E1 15338.81,E2 15338.81} C_VEL
LIN {X 0,Y 368.262,Z 547.828,A -85,B 0,C 180,E1 15338.515,E2 15338.515} C_VEL
LIN {X 0,Y 371.666,Z 526.335,A -85,B 0,C 180,E1 15338.477,E2 15338.477} C_VEL
LIN {X 0,Y 363.289,Z 509.082,A -85,B 0,C 180,E1 15336.328,E2 15336.328} C_VEL
LIN {X 0,Y 361.327,Z 503.887,A -85,B 0,C 180,E1 15335.723,E2 15335.723} C_VEL
LIN {X 0,Y 359.078,Z 485.135,A -85,B 0,C 180,E1 15332.761,E2 15332.761} C_VEL
LIN {X 0,Y 358.935,Z 470.221,A -85,B 0,C 180,E1 15330.558,E2 15330.558} C_VEL
LIN {X 0,Y 345.457,Z 477.753,A -85,B 0,C 180,E1 15329.093,E2 15329.093} C_VEL
LIN {X 0,Y 340.855,Z 480.368,A -85,B 0,C 180,E1 15328.563,E2 15328.563} C_VEL
LIN {X 0,Y 336.091,Z 483.325,A -85,B 0,C 180,E1 15328.037,E2 15328.037} C_VEL
LIN {X 0,Y 334.125,Z 484.093,A -85,B 0,C 180,E1 15327.707,E2 15327.707} C_VEL
LIN {X 0,Y 330.374,Z 522.519,A -85,B 0,C 180,E1 15324.114,E2 15324.114} C_VEL
LIN {X 0,Y 326.318,Z 541.277,A -85,B 0,C 180,E1 15322.87,E2 15322.87} C_VEL
LIN {X 0,Y 320.362,Z 627.642,A -85,B 0,C 180,E1 15319.852,E2 15319.852} C_VEL
LIN {X 0,Y 319.786,Z 654.156,A -85,B 0,C 180,E1 15318.78,E2 15318.78} C_VEL
LIN {X 0,Y 319.215,Z 668.625,A -85,B 0,C 180,E1 15317.875,E2 15317.875} C_VEL
LIN {X 0,Y 318.205,Z 683.182,A -85,B 0,C 180,E1 15316.614,E2 15316.614} C_VEL
LIN {X 0,Y 317.007,Z 695.757,A -85,B 0,C 180,E1 15315.171,E2 15315.171} C_VEL
LIN {X 0,Y 315.566,Z 707.221,A -85,B 0,C 180,E1 15313.466,E2 15313.466} C_VEL
LIN {X 0,Y 314.058,Z 717.164,A -85,B 0,C 180,E1 15311.57,E2 15311.57} C_VEL
LIN {X 0,Y 312.474,Z 725.894,A -85,B 0,C 180,E1 15309.391,E2 15309.391} C_VEL
LIN {X 0,Y 311.067,Z 732.451,A -85,B 0,C 180,E1 15307.201,E2 15307.201} C_VEL
LIN {X 0,Y 309.793,Z 737.613,A -85,B 0,C 180,E1 15304.813,E2 15304.813} C_VEL
LIN {X 0,Y 308.704,Z 741.116,A -85,B 0,C 180,E1 15302.227,E2 15302.227} C_VEL
LIN {X 0,Y 307.84,Z 742.717,A -85,B 0,C 180,E1 15299.441,E2 15299.441} C_VEL
LIN {X 0,Y 307.306,Z 742.281,A -85,B 0,C 180,E1 15296.829,E2 15296.829} C_VEL
LIN {X 0,Y 307.027,Z 740.238,A -85,B 0,C 180,E1 15294.393,E2 15294.393} C_VEL
LIN {X 0,Y 306.966,Z 736.22,A -85,B 0,C 180,E1 15291.759,E2 15291.759} C_VEL
LIN {X 0,Y 307.144,Z 730.13,A -85,B 0,C 180,E1 15289.116,E2 15289.116} C_VEL
LIN {X 0,Y 307.555,Z 722.316,A -85,B 0,C 180,E1 15286.654,E2 15286.654} C_VEL
LIN {X 0,Y 308.15,Z 712.873,A -85,B 0,C 180,E1 15284.376,E2 15284.376} C_VEL
LIN {X 0,Y 308.88,Z 701.784,A -85,B 0,C 180,E1 15282.284,E2 15282.284} C_VEL
LIN {X 0,Y 309.643,Z 689.594,A -85,B 0,C 180,E1 15280.475,E2 15280.475} C_VEL
LIN {X 0,Y 310.362,Z 676.478,A -85,B 0,C 180,E1 15278.948,E2 15278.948} C_VEL
LIN {X 0,Y 310.975,Z 662.594,A -85,B 0,C 180,E1 15277.703,E2 15277.703} C_VEL
LIN {X 0,Y 311.442,Z 647.135,A -85,B 0,C 180,E1 15276.693,E2 15276.693} C_VEL
LIN {X 0,Y 311.633,Z 631.071,A -85,B 0,C 180,E1 15276.005,E2 15276.005} C_VEL
LIN {X 0,Y 312.968,Z 570.931,A -85,B 0,C 180,E1 15274.227,E2 15274.227} C_VEL
LIN {X 0,Y 314.849,Z 519.243,A -85,B 0,C 180,E1 15272.684,E2 15272.684} C_VEL
LIN {X 0,Y 315.01,Z 518.685,A -85,B 0,C 180,E1 15272.597,E2 15272.597} C_VEL
LIN {X 0,Y 316.186,Z 518.296,A -85,B 0,C 180,E1 15272.187,E2 15272.187} C_VEL
LIN {X 0,Y 318.923,Z 514.63,A -85,B 0,C 180,E1 15271.489,E2 15271.489} C_VEL
LIN {X 0,Y 324.023,Z 505.573,A -85,B 0,C 180,E1 15270.414,E2 15270.414} C_VEL
LIN {X 0,Y 325.785,Z 502.001,A -85,B 0,C 180,E1 15270.084,E2 15270.084} C_VEL
LIN {X 0,Y 328.709,Z 499.402,A -85,B 0,C 180,E1 15269.318,E2 15269.318} C_VEL
LIN {X 0,Y 332.519,Z 493.942,A -85,B 0,C 180,E1 15268.502,E2 15268.502} C_VEL
LIN {X 0,Y 336.329,Z 487.113,A -85,B 0,C 180,E1 15267.799,E2 15267.799} C_VEL
LIN {X 0,Y 340.266,Z 483.061,A -85,B 0,C 180,E1 15266.918,E2 15266.918} C_VEL
LIN {X 0,Y 344.975,Z 476.037,A -85,B 0,C 180,E1 15266.036,E2 15266.036} C_VEL
LIN {X 0,Y 347.431,Z 471.929,A -85,B 0,C 180,E1 15265.612,E2 15265.612} C_VEL
LIN {X 0,Y 352.081,Z 466.948,A -85,B 0,C 180,E1 15264.695,E2 15264.695} C_VEL
LIN {X 0,Y 357.311,Z 459.189,A -85,B 0,C 180,E1 15263.811,E2 15263.811} C_VEL
LIN {X 0,Y 358.889,Z 456.887,A -85,B 0,C 180,E1 15263.55,E2 15263.55} C_VEL
LIN {X 0,Y 364.26,Z 451.021,A -85,B 0,C 180,E1 15262.604,E2 15262.604} C_VEL
LIN {X 0,Y 369.371,Z 443.723,A -85,B 0,C 180,E1 15261.808,E2 15261.808} C_VEL
LIN {X 0,Y 364.409,Z 498.604,A -85,B 0,C 180,E1 15260.452,E2 15260.452} C_VEL
LIN {X 0,Y 357.91,Z 555.972,A -85,B 0,C 180,E1 15258.78,E2 15258.78} C_VEL
LIN {X 0,Y 352.917,Z 597.521,A -85,B 0,C 180,E1 15257.332,E2 15257.332} C_VEL
LIN {X 0,Y 350.203,Z 618.049,A -85,B 0,C 180,E1 15256.367,E2 15256.367} C_VEL
LIN {X 0,Y 346.885,Z 637.429,A -85,B 0,C 180,E1 15255.16,E2 15255.16} C_VEL
LIN {X 0,Y 343.004,Z 655.975,A -85,B 0,C 180,E1 15253.699,E2 15253.699} C_VEL
LIN {X 0,Y 338.466,Z 674.464,A -85,B 0,C 180,E1 15251.885,E2 15251.885} C_VEL
LIN {X 0,Y 333.651,Z 691.881,A -85,B 0,C 180,E1 15249.777,E2 15249.777} C_VEL
LIN {X 0,Y 328.689,Z 708.217,A -85,B 0,C 180,E1 15247.364,E2 15247.364} C_VEL
LIN {X 0,Y 323.761,Z 723.425,A -85,B 0,C 180,E1 15244.628,E2 15244.628} C_VEL
LIN {X 0,Y 319.323,Z 736.647,A -85,B 0,C 180,E1 15241.739,E2 15241.739} C_VEL
LIN {X 0,Y 315.216,Z 748.757,A -85,B 0,C 180,E1 15238.52,E2 15238.52} C_VEL
LIN {X 0,Y 311.712,Z 759.369,A -85,B 0,C 180,E1 15235.05,E2 15235.05} C_VEL
LIN {X 0,Y 308.962,Z 768.185,A -85,B 0,C 180,E1 15231.45,E2 15231.45} C_VEL
LIN {X 0,Y 307.005,Z 775.144,A -85,B 0,C 180,E1 15227.827,E2 15227.827} C_VEL
LIN {X 0,Y 305.693,Z 780.651,A -85,B 0,C 180,E1 15224.007,E2 15224.007} C_VEL
LIN {X 0,Y 304.965,Z 784.416,A -85,B 0,C 180,E1 15220.198,E2 15220.198} C_VEL
LIN {X 0,Y 304.64,Z 786.523,A -85,B 0,C 180,E1 15216.407,E2 15216.407} C_VEL
LIN {X 0,Y 304.548,Z 787.05,A -85,B 0,C 180,E1 15212.823,E2 15212.823} C_VEL
LIN {X 0,Y 304.624,Z 786.167,A -85,B 0,C 180,E1 15209.281,E2 15209.281} C_VEL
LIN {X 0,Y 303.71,Z 785.545,A -85,B 0,C 180,E1 15207.834,E2 15207.834} C_VEL
LIN {X 0,Y 299.383,Z 783.964,A -85,B 0,C 180,E1 15205.093,E2 15205.093} C_VEL
LIN {X 0,Y 297.512,Z 782.386,A -85,B 0,C 180,E1 15203.326,E2 15203.326} C_VEL
LIN {X 0,Y 297.437,Z 781.662,A -85,B 0,C 180,E1 15202.696,E2 15202.696} C_VEL
LIN {X 0,Y 298.539,Z 776.471,A -85,B 0,C 180,E1 15198.909,E2 15198.909} C_VEL
LIN {X 0,Y 300.317,Z 769.568,A -85,B 0,C 180,E1 15195.146,E2 15195.146} C_VEL
LIN {X 0,Y 302.79,Z 761.068,A -85,B 0,C 180,E1 15191.518,E2 15191.518} C_VEL
LIN {X 0,Y 306.085,Z 750.567,A -85,B 0,C 180,E1 15187.935,E2 15187.935} C_VEL
LIN {X 0,Y 310.009,Z 738.51,A -85,B 0,C 180,E1 15184.598,E2 15184.598} C_VEL
LIN {X 0,Y 314.161,Z 725.776,A -85,B 0,C 180,E1 15181.692,E2 15181.692} C_VEL
LIN {X 0,Y 318.607,Z 711.712,A -85,B 0,C 180,E1 15179.025,E2 15179.025} C_VEL
LIN {X 0,Y 323.256,Z 696.236,A -85,B 0,C 180,E1 15176.594,E2 15176.594} C_VEL
LIN {X 0,Y 327.947,Z 679.163,A -85,B 0,C 180,E1 15174.385,E2 15174.385} C_VEL
LIN {X 0,Y 332.217,Z 661.934,A -85,B 0,C 180,E1 15172.558,E2 15172.558} C_VEL
LIN {X 0,Y 336.096,Z 644.022,A -85,B 0,C 180,E1 15171.009,E2 15171.009} C_VEL
LIN {X 0,Y 339.493,Z 625.263,A -85,B 0,C 180,E1 15169.712,E2 15169.712} C_VEL
LIN {X 0,Y 342.34,Z 605.237,A -85,B 0,C 180,E1 15168.644,E2 15168.644} C_VEL
LIN {X 0,Y 346.497,Z 569.282,A -85,B 0,C 180,E1 15167.266,E2 15167.266} C_VEL
LIN {X 0,Y 353.142,Z 512.211,A -85,B 0,C 180,E1 15165.498,E2 15165.498} C_VEL
LIN {X 0,Y 358.447,Z 456.267,A -85,B 0,C 180,E1 15164.03,E2 15164.03} C_VEL
LIN {X 0,Y 362.141,Z 403.405,A -85,B 0,C 180,E1 15162.869,E2 15162.869} C_VEL
LIN {X 0,Y 363.036,Z 384.856,A -85,B 0,C 180,E1 15162.468,E2 15162.468} C_VEL
LIN {X 0,Y 354.912,Z 373.83,A -85,B 0,C 180,E1 15160.389,E2 15160.389} C_VEL
LIN {X 0,Y 351.512,Z 365.55,A -85,B 0,C 180,E1 15157.703,E2 15157.703} C_VEL
LIN {X 0,Y 348.165,Z 368.075,A -85,B 0,C 180,E1 15157.091,E2 15157.091} C_VEL
LIN {X 0,Y 341.44,Z 373.484,A -85,B 0,C 180,E1 15155.851,E2 15155.851} C_VEL
LIN {X 0,Y 336.249,Z 377.676,A -85,B 0,C 180,E1 15154.816,E2 15154.816} C_VEL
LIN {X 0,Y 331.511,Z 381.974,A -85,B 0,C 180,E1 15153.916,E2 15153.916} C_VEL
LIN {X 0,Y 329.074,Z 383.936,A -85,B 0,C 180,E1 15153.364,E2 15153.364} C_VEL
LIN {X 0,Y 325.033,Z 387.825,A -85,B 0,C 180,E1 15152.571,E2 15152.571} C_VEL
LIN {X 0,Y 322.804,Z 389.501,A -85,B 0,C 180,E1 15151.983,E2 15151.983} C_VEL
LIN {X 0,Y 319.105,Z 393.939,A -85,B 0,C 180,E1 15151.237,E2 15151.237} C_VEL
LIN {X 0,Y 317.084,Z 396.124,A -85,B 0,C 180,E1 15150.615,E2 15150.615} C_VEL
LIN {X 0,Y 316.486,Z 396.236,A -85,B 0,C 180,E1 15150.393,E2 15150.393} C_VEL
LIN {X 0,Y 313.468,Z 442.026,A -85,B 0,C 180,E1 15145.811,E2 15145.811} C_VEL
LIN {X 0,Y 311.719,Z 466.984,A -85,B 0,C 180,E1 15143.337,E2 15143.337} C_VEL
LIN {X 0,Y 311.087,Z 471.221,A -85,B 0,C 180,E1 15143.012,E2 15143.012} C_VEL
LIN {X 0,Y 305.942,Z 603.851,A -85,B 0,C 180,E1 15138.891,E2 15138.891} C_VEL
LIN {X 0,Y 305.594,Z 623.342,A -85,B 0,C 180,E1 15138.14,E2 15138.14} C_VEL
LIN {X 0,Y 304.996,Z 640.215,A -85,B 0,C 180,E1 15137.161,E2 15137.161} C_VEL
LIN {X 0,Y 304.089,Z 657.902,A -85,B 0,C 180,E1 15135.74,E2 15135.74} C_VEL
LIN {X 0,Y 303.021,Z 674.795,A -85,B 0,C 180,E1 15133.939,E2 15133.939} C_VEL
LIN {X 0,Y 301.905,Z 690.037,A -85,B 0,C 180,E1 15131.85,E2 15131.85} C_VEL
LIN {X 0,Y 300.898,Z 703.244,A -85,B 0,C 180,E1 15129.565,E2 15129.565} C_VEL
LIN {X 0,Y 300.124,Z 713.896,A -85,B 0,C 180,E1 15127.274,E2 15127.274} C_VEL
LIN {X 0,Y 299.509,Z 723.857,A -85,B 0,C 180,E1 15124.596,E2 15124.596} C_VEL
LIN {X 0,Y 299.153,Z 732.08,A -85,B 0,C 180,E1 15121.724,E2 15121.724} C_VEL
LIN {X 0,Y 299.078,Z 737.81,A -85,B 0,C 180,E1 15119.043,E2 15119.043} C_VEL
LIN {X 0,Y 299.275,Z 742.123,A -85,B 0,C 180,E1 15116.169,E2 15116.169} C_VEL
LIN {X 0,Y 299.749,Z 744.538,A -85,B 0,C 180,E1 15113.296,E2 15113.296} C_VEL
LIN {X 0,Y 300.515,Z 745.2,A -85,B 0,C 180,E1 15110.425,E2 15110.425} C_VEL
LIN {X 0,Y 301.614,Z 743.947,A -85,B 0,C 180,E1 15107.557,E2 15107.557} C_VEL
LIN {X 0,Y 302.961,Z 741.106,A -85,B 0,C 180,E1 15104.888,E2 15104.888} C_VEL
LIN {X 0,Y 304.75,Z 736.005,A -85,B 0,C 180,E1 15102.038,E2 15102.038} C_VEL
LIN {X 0,Y 306.623,Z 729.693,A -85,B 0,C 180,E1 15099.58,E2 15099.58} C_VEL
LIN {X 0,Y 308.795,Z 721.347,A -85,B 0,C 180,E1 15097.136,E2 15097.136} C_VEL
LIN {X 0,Y 311.014,Z 711.316,A -85,B 0,C 180,E1 15094.891,E2 15094.891} C_VEL
LIN {X 0,Y 313.064,Z 700.795,A -85,B 0,C 180,E1 15093.008,E2 15093.008} C_VEL
LIN {X 0,Y 315.264,Z 687.2,A -85,B 0,C 180,E1 15091.085,E2 15091.085} C_VEL
LIN {X 0,Y 317.25,Z 671.98,A -85,B 0,C 180,E1 15089.404,E2 15089.404} C_VEL
LIN {X 0,Y 318.917,Z 655.406,A -85,B 0,C 180,E1 15088.006,E2 15088.006} C_VEL
LIN {X 0,Y 320.144,Z 638.005,A -85,B 0,C 180,E1 15086.917,E2 15086.917} C_VEL
LIN {X 0,Y 322.403,Z 608.526,A -85,B 0,C 180,E1 15085.53,E2 15085.53} C_VEL
LIN {X 0,Y 325.173,Z 606,A -85,B 0,C 180,E1 15085.165,E2 15085.165} C_VEL
LIN {X 0,Y 329.063,Z 599.785,A -85,B 0,C 180,E1 15084.835,E2 15084.835} C_VEL
LIN {X 0,Y 333.707,Z 589.652,A -85,B 0,C 180,E1 15084.602,E2 15084.602} C_VEL
LIN {X 0,Y 337.698,Z 583.931,A -85,B 0,C 180,E1 15084.181,E2 15084.181} C_VEL
LIN {X 0,Y 342.33,Z 574.4,A -85,B 0,C 180,E1 15083.83,E2 15083.83} C_VEL
LIN {X 0,Y 346.773,Z 562.744,A -85,B 0,C 180,E1 15083.562,E2 15083.562} C_VEL
LIN {X 0,Y 351.304,Z 554.217,A -85,B 0,C 180,E1 15083.081,E2 15083.081} C_VEL
LIN {X 0,Y 356.169,Z 541.283,A -85,B 0,C 180,E1 15082.648,E2 15082.648} C_VEL
LIN {X 0,Y 361.253,Z 524.468,A -85,B 0,C 180,E1 15082.24,E2 15082.24} C_VEL
LIN {X 0,Y 362.927,Z 521.298,A -85,B 0,C 180,E1 15082.039,E2 15082.039} C_VEL
LIN {X 0,Y 358.648,Z 549.67,A -85,B 0,C 180,E1 15081.937,E2 15081.937} C_VEL
LIN {X 0,Y 355.479,Z 573.168,A -85,B 0,C 180,E1 15081.543,E2 15081.543} C_VEL
LIN {X 0,Y 351.528,Z 603.94,A -85,B 0,C 180,E1 15080.552,E2 15080.552} C_VEL
LIN {X 0,Y 346.788,Z 631.829,A -85,B 0,C 180,E1 15079.377,E2 15079.377} C_VEL
LIN {X 0,Y 341.91,Z 657.559,A -85,B 0,C 180,E1 15077.959,E2 15077.959} C_VEL
LIN {X 0,Y 336.615,Z 682.783,A -85,B 0,C 180,E1 15076.203,E2 15076.203} C_VEL
LIN {X 0,Y 331.348,Z 706.314,A -85,B 0,C 180,E1 15074.191,E2 15074.191} C_VEL
LIN {X 0,Y 326.634,Z 725.155,A -85,B 0,C 180,E1 15072.203,E2 15072.203} C_VEL
LIN {X 0,Y 321.764,Z 742.839,A -85,B 0,C 180,E1 15069.918,E2 15069.918} C_VEL
LIN {X 0,Y 316.818,Z 759.378,A -85,B 0,C 180,E1 15067.297,E2 15067.297} C_VEL
LIN {X 0,Y 312.279,Z 773.953,A -85,B 0,C 180,E1 15064.522,E2 15064.522} C_VEL
LIN {X 0,Y 307.941,Z 787.673,A -85,B 0,C 180,E1 15061.358,E2 15061.358} C_VEL
LIN {X 0,Y 304.006,Z 800.466,A -85,B 0,C 180,E1 15057.783,E2 15057.783} C_VEL
LIN {X 0,Y 300.942,Z 811.135,A -85,B 0,C 180,E1 15054.121,E2 15054.121} C_VEL
LIN {X 0,Y 298.625,Z 820.46,A -85,B 0,C 180,E1 15050.174,E2 15050.174} C_VEL
LIN {X 0,Y 297.191,Z 827.84,A -85,B 0,C 180,E1 15046.215,E2 15046.215} C_VEL
LIN {X 0,Y 296.452,Z 833.797,A -85,B 0,C 180,E1 15042.016,E2 15042.016} C_VEL
LIN {X 0,Y 296.281,Z 837.695,A -85,B 0,C 180,E1 15038.148,E2 15038.148} C_VEL
LIN {X 0,Y 296.349,Z 840.084,A -85,B 0,C 180,E1 15034.257,E2 15034.257} C_VEL
LIN {X 0,Y 296.413,Z 840.998,A -85,B 0,C 180,E1 15030.58,E2 15030.58} C_VEL
LIN {X 0,Y 296.369,Z 840.606,A -85,B 0,C 180,E1 15026.906,E2 15026.906} C_VEL
LIN {X 0,Y 296.276,Z 838.79,A -85,B 0,C 180,E1 15023.022,E2 15023.022} C_VEL
LIN {X 0,Y 296.349,Z 835.384,A -85,B 0,C 180,E1 15019.053,E2 15019.053} C_VEL
LIN {X 0,Y 296.932,Z 829.992,A -85,B 0,C 180,E1 15014.772,E2 15014.772} C_VEL
LIN {X 0,Y 298.194,Z 823.312,A -85,B 0,C 180,E1 15010.816,E2 15010.816} C_VEL
LIN {X 0,Y 300.443,Z 814.342,A -85,B 0,C 180,E1 15006.67,E2 15006.67} C_VEL
LIN {X 0,Y 303.412,Z 804.335,A -85,B 0,C 180,E1 15002.95,E2 15002.95} C_VEL
LIN {X 0,Y 307.518,Z 791.655,A -85,B 0,C 180,E1 14999.132,E2 14999.132} C_VEL
LIN {X 0,Y 311.954,Z 778.478,A -85,B 0,C 180,E1 14995.881,E2 14995.881} C_VEL
LIN {X 0,Y 317.156,Z 762.994,A -85,B 0,C 180,E1 14992.75,E2 14992.75} C_VEL
LIN {X 0,Y 322.157,Z 747.502,A -85,B 0,C 180,E1 14990.163,E2 14990.163} C_VEL
LIN {X 0,Y 327.588,Z 729.463,A -85,B 0,C 180,E1 14987.7,E2 14987.7} C_VEL
LIN {X 0,Y 332.528,Z 711.447,A -85,B 0,C 180,E1 14985.694,E2 14985.694} C_VEL
LIN {X 0,Y 337.985,Z 688.878,A -85,B 0,C 180,E1 14983.672,E2 14983.672} C_VEL
LIN {X 0,Y 343.478,Z 664.64,A -85,B 0,C 180,E1 14981.898,E2 14981.898} C_VEL
LIN {X 0,Y 348.693,Z 639.367,A -85,B 0,C 180,E1 14980.42,E2 14980.42} C_VEL
LIN {X 0,Y 353.796,Z 611.859,A -85,B 0,C 180,E1 14979.182,E2 14979.182} C_VEL
LIN {X 0,Y 357.966,Z 584.016,A -85,B 0,C 180,E1 14978.209,E2 14978.209} C_VEL
LIN {X 0,Y 360.631,Z 564.453,A -85,B 0,C 180,E1 14977.733,E2 14977.733} C_VEL
LIN {X 0,Y 364.215,Z 540.806,A -85,B 0,C 180,E1 14977.517,E2 14977.517} C_VEL
LIN {X 0,Y 366.049,Z 529.072,A -85,B 0,C 180,E1 14977.501,E2 14977.501} C_VEL
LIN {X 0,Y 358.27,Z 512.234,A -85,B 0,C 180,E1 14975.386,E2 14975.386} C_VEL
LIN {X 0,Y 353.752,Z 499.735,A -85,B 0,C 180,E1 14973.932,E2 14973.932} C_VEL
LIN {X 0,Y 352.593,Z 479.53,A -85,B 0,C 180,E1 14970.769,E2 14970.769} C_VEL
LIN {X 0,Y 339.011,Z 487.298,A -85,B 0,C 180,E1 14969.313,E2 14969.313} C_VEL
LIN {X 0,Y 335.432,Z 489.609,A -85,B 0,C 180,E1 14968.874,E2 14968.874} C_VEL
LIN {X 0,Y 334.414,Z 490.881,A -85,B 0,C 180,E1 14968.628,E2 14968.628} C_VEL
LIN {X 0,Y 329.5,Z 500.927,A -85,B 0,C 180,E1 14967.564,E2 14967.564} C_VEL
LIN {X 0,Y 326.641,Z 505.394,A -85,B 0,C 180,E1 14966.839,E2 14966.839} C_VEL
LIN {X 0,Y 324.656,Z 524.248,A -85,B 0,C 180,E1 14965.053,E2 14965.053} C_VEL
LIN {X 0,Y 320.346,Z 543.406,A -85,B 0,C 180,E1 14963.779,E2 14963.779} C_VEL
LIN {X 0,Y 313.975,Z 627.953,A -85,B 0,C 180,E1 14960.724,E2 14960.724} C_VEL
LIN {X 0,Y 313.173,Z 655.706,A -85,B 0,C 180,E1 14959.549,E2 14959.549} C_VEL
LIN {X 0,Y 312.471,Z 670.877,A -85,B 0,C 180,E1 14958.565,E2 14958.565} C_VEL
LIN {X 0,Y 311.452,Z 684.353,A -85,B 0,C 180,E1 14957.37,E2 14957.37} C_VEL
LIN {X 0,Y 310.134,Z 696.891,A -85,B 0,C 180,E1 14955.904,E2 14955.904} C_VEL
LIN {X 0,Y 308.487,Z 708.997,A -85,B 0,C 180,E1 14954.068,E2 14954.068} C_VEL
LIN {X 0,Y 306.77,Z 719.274,A -85,B 0,C 180,E1 14952.039,E2 14952.039} C_VEL
LIN {X 0,Y 305.056,Z 727.849,A -85,B 0,C 180,E1 14949.813,E2 14949.813} C_VEL
LIN {X 0,Y 303.426,Z 734.775,A -85,B 0,C 180,E1 14947.383,E2 14947.383} C_VEL
LIN {X 0,Y 302.052,Z 739.626,A -85,B 0,C 180,E1 14944.937,E2 14944.937} C_VEL
LIN {X 0,Y 300.963,Z 742.721,A -85,B 0,C 180,E1 14942.475,E2 14942.475} C_VEL
LIN {X 0,Y 300.072,Z 744.176,A -85,B 0,C 180,E1 14939.808,E2 14939.808} C_VEL
LIN {X 0,Y 299.464,Z 743.752,A -85,B 0,C 180,E1 14937.116,E2 14937.116} C_VEL
LIN {X 0,Y 299.14,Z 741.739,A -85,B 0,C 180,E1 14934.629,E2 14934.629} C_VEL
LIN {X 0,Y 299.041,Z 737.721,A -85,B 0,C 180,E1 14931.927,E2 14931.927} C_VEL
LIN {X 0,Y 299.196,Z 731.626,A -85,B 0,C 180,E1 14929.213,E2 14929.213} C_VEL
LIN {X 0,Y 299.601,Z 723.828,A -85,B 0,C 180,E1 14926.686,E2 14926.686} C_VEL
LIN {X 0,Y 300.235,Z 713.976,A -85,B 0,C 180,E1 14924.249,E2 14924.249} C_VEL
LIN {X 0,Y 300.987,Z 702.808,A -85,B 0,C 180,E1 14922.104,E2 14922.104} C_VEL
LIN {X 0,Y 301.797,Z 690.177,A -85,B 0,C 180,E1 14920.204,E2 14920.204} C_VEL
LIN {X 0,Y 302.57,Z 676.289,A -85,B 0,C 180,E1 14918.582,E2 14918.582} C_VEL
LIN {X 0,Y 303.206,Z 661.869,A -85,B 0,C 180,E1 14917.304,E2 14917.304} C_VEL
LIN {X 0,Y 303.661,Z 646.236,A -85,B 0,C 180,E1 14916.306,E2 14916.306} C_VEL
LIN {X 0,Y 303.835,Z 629.78,A -85,B 0,C 180,E1 14915.632,E2 14915.632} C_VEL
LIN {X 0,Y 305.396,Z 566.761,A -85,B 0,C 180,E1 14913.71,E2 14913.71} C_VEL
LIN {X 0,Y 306.077,Z 549.889,A -85,B 0,C 180,E1 14913.152,E2 14913.152} C_VEL
LIN {X 0,Y 306.931,Z 549.861,A -85,B 0,C 180,E1 14912.813,E2 14912.813} C_VEL
LIN {X 0,Y 308.711,Z 547.222,A -85,B 0,C 180,E1 14912.382,E2 14912.382} C_VEL
LIN {X 0,Y 311.721,Z 540.245,A -85,B 0,C 180,E1 14911.908,E2 14911.908} C_VEL
LIN {X 0,Y 315.876,Z 527.665,A -85,B 0,C 180,E1 14911.504,E2 14911.504} C_VEL
LIN {X 0,Y 316.705,Z 525.091,A -85,B 0,C 180,E1 14911.425,E2 14911.425} C_VEL
LIN {X 0,Y 320.029,Z 520.907,A -85,B 0,C 180,E1 14910.599,E2 14910.599} C_VEL
LIN {X 0,Y 325.888,Z 510.971,A -85,B 0,C 180,E1 14909.407,E2 14909.407} C_VEL
LIN {X 0,Y 327.368,Z 508.305,A -85,B 0,C 180,E1 14909.128,E2 14909.128} C_VEL
LIN {X 0,Y 331.258,Z 504.189,A -85,B 0,C 180,E1 14908.216,E2 14908.216} C_VEL
LIN {X 0,Y 335.862,Z 497.212,A -85,B 0,C 180,E1 14907.319,E2 14907.319} C_VEL
LIN {X 0,Y 338.224,Z 493.18,A -85,B 0,C 180,E1 14906.895,E2 14906.895} C_VEL
LIN {X 0,Y 342.822,Z 488.146,A -85,B 0,C 180,E1 14905.945,E2 14905.945} C_VEL
LIN {X 0,Y 348.029,Z 480.318,A -85,B 0,C 180,E1 14905.029,E2 14905.029} C_VEL
LIN {X 0,Y 349.608,Z 477.899,A -85,B 0,C 180,E1 14904.76,E2 14904.76} C_VEL
LIN {X 0,Y 354.91,Z 472.006,A -85,B 0,C 180,E1 14903.777,E2 14903.777} C_VEL
LIN {X 0,Y 361.149,Z 462.96,A -85,B 0,C 180,E1 14902.775,E2 14902.775} C_VEL
LIN {X 0,Y 363.173,Z 461.03,A -85,B 0,C 180,E1 14902.416,E2 14902.416} C_VEL
LIN {X 0,Y 357.698,Z 515.306,A -85,B 0,C 180,E1 14900.995,E2 14900.995} C_VEL
LIN {X 0,Y 350.448,Z 574.022,A -85,B 0,C 180,E1 14899.182,E2 14899.182} C_VEL
LIN {X 0,Y 346.267,Z 607.835,A -85,B 0,C 180,E1 14897.865,E2 14897.865} C_VEL
LIN {X 0,Y 343.114,Z 628.107,A -85,B 0,C 180,E1 14896.763,E2 14896.763} C_VEL
LIN {X 0,Y 339.231,Z 647.642,A -85,B 0,C 180,E1 14895.383,E2 14895.383} C_VEL
LIN {X 0,Y 334.816,Z 666.252,A -85,B 0,C 180,E1 14893.723,E2 14893.723} C_VEL
LIN {X 0,Y 330.052,Z 683.752,A -85,B 0,C 180,E1 14891.796,E2 14891.796} C_VEL
LIN {X 0,Y 325.011,Z 700.399,A -85,B 0,C 180,E1 14889.555,E2 14889.555} C_VEL
LIN {X 0,Y 319.804,Z 716.211,A -85,B 0,C 180,E1 14886.956,E2 14886.956} C_VEL
LIN {X 0,Y 314.681,Z 730.918,A -85,B 0,C 180,E1 14884.002,E2 14884.002} C_VEL
LIN {X 0,Y 310.084,Z 743.769,A -85,B 0,C 180,E1 14880.844,E2 14880.844} C_VEL
LIN {X 0,Y 306.044,Z 755.106,A -85,B 0,C 180,E1 14877.43,E2 14877.43} C_VEL
LIN {X 0,Y 302.701,Z 764.82,A -85,B 0,C 180,E1 14873.797,E2 14873.797} C_VEL
LIN {X 0,Y 300.186,Z 772.723,A -85,B 0,C 180,E1 14870.064,E2 14870.064} C_VEL
LIN {X 0,Y 298.396,Z 779.066,A -85,B 0,C 180,E1 14866.148,E2 14866.148} C_VEL
LIN {X 0,Y 297.343,Z 783.615,A -85,B 0,C 180,E1 14862.231,E2 14862.231} C_VEL
LIN {X 0,Y 296.806,Z 786.471,A -85,B 0,C 180,E1 14858.329,E2 14858.329} C_VEL
LIN {X 0,Y 296.601,Z 787.706,A -85,B 0,C 180,E1 14854.447,E2 14854.447} C_VEL
LIN {X 0,Y 296.601,Z 787.414,A -85,B 0,C 180,E1 14850.773,E2 14850.773} C_VEL
LIN {X 0,Y 296.799,Z 785.705,A -85,B 0,C 180,E1 14847.104,E2 14847.104} C_VEL
LIN {X 0,Y 297.331,Z 782.311,A -85,B 0,C 180,E1 14843.241,E2 14843.241} C_VEL
LIN {X 0,Y 297.437,Z 781.662,A -85,B 0,C 180,E1 14842.696,E2 14842.696} C_VEL
LIN {X 0,Y 296.798,Z 780.033,A -85,B 0,C 180,E1 14841.24,E2 14841.24} C_VEL
LIN {X 0,Y 291.925,Z 774.922,A -85,B 0,C 180,E1 14837.216,E2 14837.216} C_VEL
LIN {X 0,Y 291.846,Z 772.956,A -85,B 0,C 180,E1 14836.075,E2 14836.075} C_VEL
LIN {X 0,Y 294.294,Z 764.779,A -85,B 0,C 180,E1 14832.195,E2 14832.195} C_VEL
LIN {X 0,Y 297.498,Z 754.983,A -85,B 0,C 180,E1 14828.51,E2 14828.51} C_VEL
LIN {X 0,Y 301.352,Z 743.698,A -85,B 0,C 180,E1 14825.078,E2 14825.078} C_VEL
LIN {X 0,Y 305.735,Z 730.94,A -85,B 0,C 180,E1 14821.905,E2 14821.905} C_VEL
LIN {X 0,Y 310.526,Z 716.699,A -85,B 0,C 180,E1 14818.99,E2 14818.99} C_VEL
LIN {X 0,Y 315.403,Z 701.43,A -85,B 0,C 180,E1 14816.414,E2 14816.414} C_VEL
LIN {X 0,Y 320.248,Z 685.073,A -85,B 0,C 180,E1 14814.142,E2 14814.142} C_VEL
LIN {X 0,Y 324.859,Z 667.779,A -85,B 0,C 180,E1 14812.172,E2 14812.172} C_VEL
LIN {X 0,Y 328.976,Z 650.155,A -85,B 0,C 180,E1 14810.533,E2 14810.533} C_VEL
LIN {X 0,Y 332.614,Z 631.929,A -85,B 0,C 180,E1 14809.17,E2 14809.17} C_VEL
LIN {X 0,Y 335.709,Z 612.676,A -85,B 0,C 180,E1 14808.038,E2 14808.038} C_VEL
LIN {X 0,Y 338.771,Z 587.968,A -85,B 0,C 180,E1 14806.96,E2 14806.96} C_VEL
LIN {X 0,Y 345.305,Z 535.439,A -85,B 0,C 180,E1 14805.188,E2 14805.188} C_VEL
LIN {X 0,Y 351.295,Z 480.01,A -85,B 0,C 180,E1 14803.613,E2 14803.613} C_VEL
LIN {X 0,Y 355.748,Z 426.638,A -85,B 0,C 180,E1 14802.349,E2 14802.349} C_VEL
LIN {X 0,Y 357.978,Z 389.101,A -85,B 0,C 180,E1 14801.557,E2 14801.557} C_VEL
LIN {X 0,Y 348.769,Z 376.549,A -85,B 0,C 180,E1 14799.021,E2 14799.021} C_VEL
LIN {X 0,Y 347.426,Z 373.728,A -85,B 0,C 180,E1 14798.016,E2 14798.016} C_VEL
LIN {X 0,Y 339.872,Z 379.791,A -85,B 0,C 180,E1 14796.67,E2 14796.67} C_VEL
LIN {X 0,Y 333.749,Z 384.935,A -85,B 0,C 180,E1 14795.483,E2 14795.483} C_VEL
LIN {X 0,Y 329.474,Z 389.463,A -85,B 0,C 180,E1 14794.418,E2 14794.418} C_VEL
LIN {X 0,Y 324.988,Z 394.812,A -85,B 0,C 180,E1 14793.258,E2 14793.258} C_VEL
LIN {X 0,Y 323.051,Z 396.746,A -85,B 0,C 180,E1 14792.717,E2 14792.717} C_VEL
LIN {X 0,Y 318.904,Z 402.412,A -85,B 0,C 180,E1 14791.575,E2 14791.575} C_VEL
LIN {X 0,Y 317.862,Z 403.658,A -85,B 0,C 180,E1 14791.267,E2 14791.267} C_VEL
LIN {X 0,Y 313.101,Z 415.125,A -85,B 0,C 180,E1 14790.091,E2 14790.091} C_VEL
LIN {X 0,Y 309.617,Z 421.757,A -85,B 0,C 180,E1 14789.08,E2 14789.08} C_VEL
LIN {X 0,Y 307.95,Z 423.766,A -85,B 0,C 180,E1 14788.509,E2 14788.509} C_VEL
LIN {X 0,Y 307.342,Z 424.071,A -85,B 0,C 180,E1 14788.253,E2 14788.253} C_VEL
LIN {X 0,Y 304.556,Z 465.978,A -85,B 0,C 180,E1 14784.023,E2 14784.023} C_VEL
LIN {X 0,Y 303.554,Z 472.156,A -85,B 0,C 180,E1 14783.508,E2 14783.508} C_VEL
LIN {X 0,Y 298.184,Z 604.216,A -85,B 0,C 180,E1 14779.255,E2 14779.255} C_VEL
LIN {X 0,Y 297.808,Z 624.295,A -85,B 0,C 180,E1 14778.467,E2 14778.467} C_VEL
LIN {X 0,Y 297.163,Z 641.743,A -85,B 0,C 180,E1 14777.426,E2 14777.426} C_VEL
LIN {X 0,Y 296.224,Z 659.382,A -85,B 0,C 180,E1 14775.968,E2 14775.968} C_VEL
LIN {X 0,Y 295.12,Z 676.213,A -85,B 0,C 180,E1 14774.12,E2 14774.12} C_VEL
LIN {X 0,Y 293.972,Z 691.435,A -85,B 0,C 180,E1 14771.975,E2 14771.975} C_VEL
LIN {X 0,Y 292.907,Z 705.148,A -85,B 0,C 180,E1 14769.53,E2 14769.53} C_VEL
LIN {X 0,Y 292.102,Z 716.111,A -85,B 0,C 180,E1 14767.079,E2 14767.079} C_VEL
LIN {X 0,Y 291.546,Z 725.341,A -85,B 0,C 180,E1 14764.525,E2 14764.525} C_VEL
LIN {X 0,Y 291.206,Z 733.623,A -85,B 0,C 180,E1 14761.575,E2 14761.575} C_VEL
LIN {X 0,Y 291.167,Z 739.696,A -85,B 0,C 180,E1 14758.623,E2 14758.623} C_VEL
LIN {X 0,Y 291.406,Z 743.691,A -85,B 0,C 180,E1 14755.869,E2 14755.869} C_VEL
LIN {X 0,Y 291.952,Z 746.133,A -85,B 0,C 180,E1 14752.919,E2 14752.919} C_VEL
LIN {X 0,Y 292.753,Z 746.82,A -85,B 0,C 180,E1 14750.168,E2 14750.168} C_VEL
LIN {X 0,Y 293.959,Z 745.697,A -85,B 0,C 180,E1 14747.228,E2 14747.228} C_VEL
LIN {X 0,Y 295.547,Z 742.733,A -85,B 0,C 180,E1 14744.298,E2 14744.298} C_VEL
LIN {X 0,Y 297.381,Z 738.032,A -85,B 0,C 180,E1 14741.577,E2 14741.577} C_VEL
LIN {X 0,Y 299.434,Z 731.934,A -85,B 0,C 180,E1 14739.067,E2 14739.067} C_VEL
LIN {X 0,Y 301.976,Z 723.037,A -85,B 0,C 180,E1 14736.383,E2 14736.383} C_VEL
LIN {X 0,Y 304.41,Z 713.085,A -85,B 0,C 180,E1 14734.098,E2 14734.098} C_VEL
LIN {X 0,Y 306.846,Z 701.549,A -85,B 0,C 180,E1 14732.014,E2 14732.014} C_VEL
LIN {X 0,Y 309.074,Z 689.17,A -85,B 0,C 180,E1 14730.227,E2 14730.227} C_VEL
LIN {X 0,Y 311.261,Z 674.342,A -85,B 0,C 180,E1 14728.534,E2 14728.534} C_VEL
LIN {X 0,Y 313.146,Z 658.221,A -85,B 0,C 180,E1 14727.114,E2 14727.114} C_VEL
LIN {X 0,Y 314.614,Z 640.788,A -85,B 0,C 180,E1 14725.963,E2 14725.963} C_VEL
LIN {X 0,Y 315.583,Z 627.652,A -85,B 0,C 180,E1 14725.285,E2 14725.285} C_VEL
LIN {X 0,Y 318.337,Z 625.598,A -85,B 0,C 180,E1 14724.916,E2 14724.916} C_VEL
LIN {X 0,Y 322.009,Z 620.551,A -85,B 0,C 180,E1 14724.614,E2 14724.614} C_VEL
LIN {X 0,Y 326.039,Z 613.217,A -85,B 0,C 180,E1 14724.422,E2 14724.422} C_VEL
LIN {X 0,Y 330.113,Z 608.288,A -85,B 0,C 180,E1 14724.014,E2 14724.014} C_VEL
LIN {X 0,Y 334.992,Z 599.57,A -85,B 0,C 180,E1 14723.705,E2 14723.705} C_VEL
LIN {X 0,Y 337.8,Z 593.527,A -85,B 0,C 180,E1 14723.571,E2 14723.571} C_VEL
LIN {X 0,Y 342.604,Z 586.161,A -85,B 0,C 180,E1 14723.133,E2 14723.133} C_VEL
LIN {X 0,Y 347.609,Z 575.474,A -85,B 0,C 180,E1 14722.802,E2 14722.802} C_VEL
LIN {X 0,Y 350.835,Z 566.956,A -85,B 0,C 180,E1 14722.631,E2 14722.631} C_VEL
LIN {X 0,Y 347.829,Z 590.411,A -85,B 0,C 180,E1 14721.965,E2 14721.965} C_VEL
LIN {X 0,Y 343.242,Z 619.478,A -85,B 0,C 180,E1 14720.858,E2 14720.858} C_VEL
LIN {X 0,Y 338.361,Z 645.417,A -85,B 0,C 180,E1 14719.581,E2 14719.581} C_VEL
LIN {X 0,Y 332.85,Z 671.867,A -85,B 0,C 180,E1 14717.9,E2 14717.9} C_VEL
LIN {X 0,Y 327.442,Z 695.854,A -85,B 0,C 180,E1 14716.006,E2 14716.006} C_VEL
LIN {X 0,Y 322.566,Z 715.68,A -85,B 0,C 180,E1 14714.098,E2 14714.098} C_VEL
LIN {X 0,Y 317.677,Z 733.581,A -85,B 0,C 180,E1 14711.977,E2 14711.977} C_VEL
LIN {X 0,Y 312.606,Z 750.398,A -85,B 0,C 180,E1 14709.531,E2 14709.531} C_VEL
LIN {X 0,Y 307.381,Z 766.729,A -85,B 0,C 180,E1 14706.648,E2 14706.648} C_VEL
LIN {X 0,Y 302.553,Z 781.298,A -85,B 0,C 180,E1 14703.497,E2 14703.497} C_VEL
LIN {X 0,Y 298.143,Z 794.709,A -85,B 0,C 180,E1 14699.98,E2 14699.98} C_VEL
LIN {X 0,Y 294.46,Z 806.404,A -85,B 0,C 180,E1 14696.195,E2 14696.195} C_VEL
LIN {X 0,Y 291.63,Z 816.547,A -85,B 0,C 180,E1 14692.157,E2 14692.157} C_VEL
LIN {X 0,Y 289.689,Z 824.961,A -85,B 0,C 180,E1 14687.89,E2 14687.89} C_VEL
LIN {X 0,Y 288.653,Z 831.451,A -85,B 0,C 180,E1 14683.624,E2 14683.624} C_VEL
LIN {X 0,Y 288.314,Z 836.063,A -85,B 0,C 180,E1 14679.381,E2 14679.381} C_VEL
LIN {X 0,Y 288.347,Z 838.891,A -85,B 0,C 180,E1 14675.372,E2 14675.372} C_VEL
LIN {X 0,Y 288.432,Z 840.188,A -85,B 0,C 180,E1 14671.589,E2 14671.589} C_VEL
LIN {X 0,Y 288.419,Z 840.143,A -85,B 0,C 180,E1 14667.814,E2 14667.814} C_VEL
LIN {X 0,Y 288.312,Z 838.77,A -85,B 0,C 180,E1 14664.028,E2 14664.028} C_VEL
LIN {X 0,Y 288.309,Z 835.877,A -85,B 0,C 180,E1 14660.014,E2 14660.014} C_VEL
LIN {X 0,Y 288.733,Z 831.224,A -85,B 0,C 180,E1 14655.767,E2 14655.767} C_VEL
LIN {X 0,Y 289.901,Z 824.745,A -85,B 0,C 180,E1 14651.5,E2 14651.5} C_VEL
LIN {X 0,Y 292.019,Z 816.373,A -85,B 0,C 180,E1 14647.238,E2 14647.238} C_VEL
LIN {X 0,Y 295.057,Z 806.357,A -85,B 0,C 180,E1 14643.211,E2 14643.211} C_VEL
LIN {X 0,Y 298.963,Z 794.823,A -85,B 0,C 180,E1 14639.445,E2 14639.445} C_VEL
LIN {X 0,Y 303.61,Z 781.687,A -85,B 0,C 180,E1 14635.954,E2 14635.954} C_VEL
LIN {X 0,Y 308.838,Z 766.959,A -85,B 0,C 180,E1 14632.741,E2 14632.741} C_VEL
LIN {X 0,Y 314.127,Z 751.57,A -85,B 0,C 180,E1 14629.987,E2 14629.987} C_VEL
LIN {X 0,Y 319.815,Z 733.92,A -85,B 0,C 180,E1 14627.398,E2 14627.398} C_VEL
LIN {X 0,Y 325.028,Z 716.197,A -85,B 0,C 180,E1 14625.284,E2 14625.284} C_VEL
LIN {X 0,Y 329.935,Z 697.303,A -85,B 0,C 180,E1 14623.465,E2 14623.465} C_VEL
LIN {X 0,Y 335.321,Z 675.059,A -85,B 0,C 180,E1 14621.677,E2 14621.677} C_VEL
LIN {X 0,Y 340.891,Z 649.965,A -85,B 0,C 180,E1 14620.045,E2 14620.045} C_VEL
LIN {X 0,Y 345.954,Z 625.096,A -85,B 0,C 180,E1 14618.774,E2 14618.774} C_VEL
LIN {X 0,Y 351.096,Z 595.711,A -85,B 0,C 180,E1 14617.613,E2 14617.613} C_VEL
LIN {X 0,Y 354.658,Z 570.186,A -85,B 0,C 180,E1 14616.857,E2 14616.857} C_VEL
LIN {X 0,Y 358.281,Z 546.728,A -85,B 0,C 180,E1 14616.55,E2 14616.55} C_VEL
LIN {X 0,Y 360.578,Z 532.014,A -85,B 0,C 180,E1 14616.508,E2 14616.508} C_VEL
LIN {X 0,Y 353.137,Z 514.649,A -85,B 0,C 180,E1 14614.343,E2 14614.343} C_VEL
LIN {X 0,Y 347.311,Z 497.774,A -85,B 0,C 180,E1 14612.375,E2 14612.375} C_VEL
LIN {X 0,Y 346.806,Z 495.07,A -85,B 0,C 180,E1 14612.037,E2 14612.037} C_VEL
LIN {X 0,Y 346.604,Z 488.769,A -85,B 0,C 180,E1 14611.044,E2 14611.044} C_VEL
LIN {X 0,Y 340.142,Z 492.568,A -85,B 0,C 180,E1 14610.322,E2 14610.322} C_VEL
LIN {X 0,Y 336.561,Z 496.972,A -85,B 0,C 180,E1 14609.504,E2 14609.504} C_VEL
LIN {X 0,Y 331.418,Z 506.995,A -85,B 0,C 180,E1 14608.419,E2 14608.419} C_VEL
LIN {X 0,Y 328.713,Z 511.468,A -85,B 0,C 180,E1 14607.784,E2 14607.784} C_VEL
LIN {X 0,Y 323.315,Z 523.839,A -85,B 0,C 180,E1 14606.641,E2 14606.641} C_VEL
LIN {X 0,Y 320.588,Z 529.803,A -85,B 0,C 180,E1 14606.047,E2 14606.047} C_VEL
LIN {X 0,Y 315.476,Z 541.518,A -85,B 0,C 180,E1 14604.981,E2 14604.981} C_VEL
LIN {X 0,Y 314.588,Z 546.33,A -85,B 0,C 180,E1 14604.729,E2 14604.729} C_VEL
LIN {X 0,Y 307.838,Z 627.205,A -85,B 0,C 180,E1 14601.7,E2 14601.7} C_VEL
LIN {X 0,Y 306.714,Z 657.136,A -85,B 0,C 180,E1 14600.383,E2 14600.383} C_VEL
LIN {X 0,Y 305.932,Z 672.367,A -85,B 0,C 180,E1 14599.373,E2 14599.373} C_VEL
LIN {X 0,Y 304.701,Z 686.58,A -85,B 0,C 180,E1 14598.064,E2 14598.064} C_VEL
LIN {X 0,Y 303.172,Z 699.599,A -85,B 0,C 180,E1 14596.476,E2 14596.476} C_VEL
